				_pTimeValue := F_BACnet_EndOf(_pDailySched, SIZEOF(ST_BACnet_SpecialEventList));
				_nTimeValue := 1;
				WHILE _pTimeValue <> 0 DO
					Sched_ReadEntry(eDatatype, _pTimeValue, tCalendar[_nCalEntry].stEntry[_nTimeValue]);
					_nTimeValue:=_nTimeValue+1;
					_pTimeValue:=F_BACnet_NextListElem(_pTimeValue, _pTimeValue^.nEntrySize);
				END_WHILE		
				_nCalEntry:=_nCalEntry+1;
			ELSE
				tException[_nExcEntry].eType := _pDailySched^.stEvent.eCalEntryChoice + 1;
				tException[_nExcEntry].uDate := _pDailySched^.stEvent.uCalEntry;
				tException[_nExcEntry].nEventPriority := _pDailySched^.stEvent.nEventPriority;
				
				_pTimeValue := F_BACnet_EndOf(_pDailySched, SIZEOF(ST_BACnet_SpecialEventList));
				_nTimeValue := 1;
				WHILE _pTimeValue <> 0 DO
					Sched_ReadEntry(eDatatype, _pTimeValue, tException[_nExcEntry].stEntry[_nTimeValue]);
					_nTimeValue:=_nTimeValue+1;
					_pTimeValue:=F_BACnet_NextListElem(_pTimeValue, _pTimeValue^.nEntrySize);
				END_WHILE					
				_nExcEntry:=_nExcEntry+1;
			END_IF
			_pDailySched:=F_BACnet_NextListElem(_pDailySched, _pDailySched^.nEntrySize);
		END_WHILE
	END_IF
END_IF

ReadPropertyExceptionSched:=_hResult;
END_METHOD

METHOD ReadPropertyLimitEnable : HRESULT
VAR CONSTANT
	ePropID : E_BACnetPropIdentifier := E_BACnetPropIdentifier.PropLimitEnable;
END_VAR
VAR_INPUT
	value : REFERENCE TO ST_BACnet_LimitEnable;
END_VAR
VAR
	_flags : WORD := 16#0006;
	_size : DINT := 2;
END_VAR
IF (ipObj <> 0) AND (__ISVALIDREF(value)) THEN
	ReadPropertyLimitEnable := ReadProperty(ePropID, ADR(_flags), ADR(_size));
	
	IF (ReadPropertyLimitEnable = S_OK) THEN
		value.highLimitEnable := _flags.14;
		value.lowLimitEnable := _flags.15;
	END_IF
ELSE
	ReadPropertyLimitEnable := E_FAIL;
END_IF
END_METHOD

METHOD ReadPropertyLogBuffer : HRESULT
VAR_IN_OUT
	tLogBuffer						: ARRAY [*] OF ST_BA_TrendEntry;
END_VAR
VAR
	_nLength						: DINT;
	_cbTotalBuf						: UDINT;
	
	_pLbRecordList					: POINTER TO ST_BACnet_LogRecordList;								// Log buffer - record list
	_pLrDatumList					: POINTER TO ST_BACnet_LogDatumList;
	_nNextRecPos					: UDINT;
	_nRecCount						: UDINT;															// Log record entry - datum list
	_nMaxSeq						: DWORD;
	
	_nRec							: UDINT;
	
	
	_stRecListTmp					: POINTER TO ST_BACnet_LogRecordList;
END_VAR
IF (ipObj = 0) THEN
	_hResult := E_FAIL;
ELSE
	_nLength := SIZEOF(BACnet_Globals.bDefaultBuffer);
	_hResult := ReadProperty(E_BACnetPropIdentifier.PropLogBuffer, ADR(BACnet_Globals.bDefaultBuffer), ADR(_nLength));
	
	IF (SUCCEEDED(_hResult)) THEN
		IF (_nLength > 0) THEN
			MEMSET(ADR(tLogBuffer), 0, TO_UDINT(F_BA_TrendBufferSize(tLogBuffer)));
			
			// Point to first data:
			_pLbRecordList := ADR(BACnet_Globals.bDefaultBuffer);
			_cbTotalBuf := 0;
			_nNextRecPos := 0;
			_nRecCount := 0;
			_nMaxSeq := 0;
			
			REPEAT
				IF ((_pLbRecordList^.nEntrySize AND 16#7FFFFFFF) > 0) THEN
	
					_stRecListTmp := _pLbRecordList;
					
(* DEBUG *)			iOwner.LogMsg.Show3(ADSLOG_MSGTYPE_ERROR, 'DBG_TLOG', 'Record= %d, SeqID=%d, Size=%d', F_UDINT(_nNextRecPos), F_UDINT(_stRecListTmp^.nSequence), F_UDINT(_stRecListTmp^.nEntrySize), TRUE);
		
		
					(*
					// Insert pointer to record entry:
					_arrRecords[_nNextRecPos] := _pLbRecordList;
					*)
					// Select next free record position and count:
					_nNextRecPos := _nNextRecPos + 1;
					_nRecCount := _nRecCount + 1;
				END_IF
	
				// Next record entry:
				IF (NOT Trend_NextLogRecord(_pLbRecordList, _cbTotalBuf)) THEN
					EXIT;
				END_IF

			UNTIL (		(_nRecCount >= (BACnet_Globals.nDataField_MaxLogBufferEntries+1)) (* result buffer full *)
					OR	(_pLbRecordList >= (ADR(BACnet_Globals.bDefaultBuffer) + _nLength)) (* ads buffer ending reached *)
				)
			END_REPEAT

			
(* DEBUG *)	iOwner.LogMsg.Show(ADSLOG_MSGTYPE_ERROR, 'DBG_TLOG', '-----------------', TRUE);

//			// Select record list entry:
//			REPEAT
//				IF ((_pLbRecordList^.nEntrySize AND 16#7FFFFFFF) > 0) THEN
//	
//					(* check sequence order *)
//					IF _nMaxSeq > _pLbRecordList^.nSequence THEN
//						(* current sequence is lower then previous one - scan entries and sort *)
//						FOR _nRec := 0 TO _nRecCount-1 DO
//							IF _arrRecords[_nRec]^.nSequence > _pLbRecordList^.nSequence THEN
//								(* found higher sequence no. - move *)
//								_nNextRecPos := _nRec; (* remind insert position *)
//								(* check free space *)
//								IF (_nRecCount-1 < BACnet_Globals.nDataField_MaxLogBufferEntries) THEN
//									(* enough space at end of list - move *)
//									MEMMOVE(	ADR(_arrRecords[_nRec+1]), (* one position up *)
//												ADR(_arrRecords[_nRec]), (* free insert position *)
//												(_nRecCount - _nRec)*SIZEOF(_arrRecords[0]) (* move all element behind insert position *)
//									);
//								END_IF
//								EXIT; (* leave *)
//							END_IF
//						END_FOR
//					ELSE
//						(* remind sequence no. *)
//						_nMaxSeq := _pLbRecordList^.nSequence;
//					END_IF
//	
//					(* insert pointer to record entry *)
//					_arrRecords[_nNextRecPos] := _pLbRecordList;
//					(* select next free record position and count *)
//					_nNextRecPos := _nNextRecPos + 1;
//					_nRecCount := _nRecCount + 1;
//				END_IF
//	
//				(* next record entry *)
//				_NextLogRecord();
//	
//			UNTIL (		(NOT _bNextRecord) (* no more record entries *)
//					OR	(_nRecCount >= (BACnet_Globals.nDataField_MaxLogBufferEntries+1)) (* result buffer full *)
//					OR	(_pLbRecordList >= (_pAdsBuf + stBACnet_AdsBuffer.iLocked)) (* ads buffer ending reached *)
//				)
//			END_REPEAT
			
		END_IF
	ELSE
		iOwner.LogMsg.Show1(ADSLOG_MSGTYPE_ERROR, 'RLB23', 'Failed to read log buffer property! (Error 0x%x)', F_DINT(_hResult), TRUE);
	END_IF
END_IF


ReadPropertyLogBuffer := _hResult;
END_METHOD

METHOD ReadPropertyNotifyType : HRESULT
VAR CONSTANT
	ePropID : E_BACnetPropIdentifier := E_BACnetPropIdentifier.PropNotifyType;
END_VAR
VAR_INPUT
	value : REFERENCE TO E_BACnet_NotifyType;
END_VAR
VAR
	_size : DINT := 4;
END_VAR
IF (ipObj <> 0) AND (__ISVALIDREF(value)) THEN
	ReadPropertyNotifyType := ReadProperty(ePropID, ADR(value), ADR(_size));
ELSE
	ReadPropertyNotifyType := E_FAIL;
END_IF
END_METHOD

METHOD ReadPropertyReal : HRESULT
VAR_INPUT
	ePropID : E_BACnetPropIdentifier;
	value : REFERENCE TO REAL;
END_VAR
VAR
	_size : DINT := 4;
END_VAR
IF (ipObj <> 0) AND (__ISVALIDREF(value)) THEN
	ReadPropertyReal := ReadProperty(ePropID, ADR(value), ADR(_size));
ELSE
	ReadPropertyReal := E_FAIL;
END_IF
END_METHOD

METHOD ReadPropertyRecipientList : HRESULT
VAR_IN_OUT
	stRecipientList			: ARRAY[*] OF ST_BACnet_Destination;
END_VAR
// [Bugworkaround]
// > _stUnused" has to be static, otherwise its memory can be initialized incorrectly by PLC :(
VAR_STAT
	_nTemp					: DINT;
	_nSize					: DINT;
	_stUnused				: ST_BACnet_Destination;
END_VAR
IF (ipObj = 0) THEN
	_hResult := E_FAIL;
ELSE
	// Reset current content:
	F_BA_MemSetArr(stRecipientList, LOWER_BOUND(stRecipientList, 1), UPPER_BOUND(stRecipientList, 1), _stUnused);
		
	_nSize := (UPPER_BOUND(stRecipientList, 1) - LOWER_BOUND(stRecipientList, 1) + 1) * SIZEOF(ST_BACnet_Destination);
	_hResult := ReadProperty(E_BACnetPropIdentifier.PropRecipientList, stRecipientList, ADR(_nSize));
END_IF

ReadPropertyRecipientList := _hResult;
END_METHOD

METHOD ReadPropertyReference : HRESULT
VAR_INPUT
	eProperty				: E_BACnetPropIdentifier;
END_VAR
VAR_IN_OUT
	stRefObject				: ST_BACnet_ObjectPropertyReference;
END_VAR
VAR
	stTemp					: ST_BACnet_DeviceObjectPropertyReference;
END_VAR
IF (ipObj <> 0) THEN
	ReadPropertyReference := ReadProperty(eProperty, ADR(stTemp), ADR(stTemp));
	
	IF (S_OK = ReadPropertyReference) THEN
		stRefObject.tObjectID := stTemp.tObjId;
		stRefObject.ePropertyId := stTemp.ePropIdentifier;
	
		// Reset previous reference.
		// > Current interface pointer has to be resolved now via PLC!
		stRefObject.iObject := 0;
	END_IF
ELSE
	ReadPropertyReference := E_FAIL;
END_IF
END_METHOD

METHOD ReadPropertyStatusFlags : HRESULT
VAR_INPUT
	stateFlags : REFERENCE TO ST_BA_StatusFlags;
END_VAR
VAR
	_flags : DWORD;
	_size : DINT := 2;
END_VAR
IF (ipObj <> 0) AND (__ISVALIDREF(stateFlags)) THEN
	ReadPropertyStatusFlags:=ReadProperty(E_BACnetPropIdentifier.PropStatusFlags, ADR(_flags), ADR(_size));
	
	IF (ReadPropertyStatusFlags = S_OK) THEN
		stateFlags.bInAlarm:= F_BACnet_IsBitFieldBitSet(_flags, E_BACnet_StatusFlags.eInAlarm);
		stateFlags.bFault:= F_BACnet_IsBitFieldBitSet(_flags, E_BACnet_StatusFlags.eFault);
		stateFlags.bOverridden:= F_BACnet_IsBitFieldBitSet(_flags, E_BACnet_StatusFlags.eOverridden);
		stateFlags.bOutOfService:= F_BACnet_IsBitFieldBitSet(_flags, E_BACnet_StatusFlags.eOutOfService);
	END_IF
ELSE
	ReadPropertyStatusFlags := E_FAIL;
END_IF
END_METHOD

METHOD ReadPropertyString : HRESULT
VAR_INPUT
	ePropID : E_BACnetPropIdentifier;
	value : REFERENCE TO T_MaxString;
END_VAR
VAR
	_size : UDINT := 255;
	_fbDecode : FB_BACnet_StringExtDecode;
END_VAR
IF (ipObj <> 0) AND (__ISVALIDREF(value)) THEN
	_size:=SIZEOF(BACnet_Globals.stADSBuffer);
	ReadPropertyString:=ReadProperty(ePropID, ADR(BACnet_Globals.stADSBuffer), ADR(_size));
	
	IF (ReadPropertyString = S_OK) THEN
		memset(ADR(value)+_size,0,1);
		_fbDecode(pChrStringExt:=ADR(BACnet_Globals.stADSBuffer), pOutString:=ADR(value), nOutSize:=_size);
		
		IF NOT _fbDecode.bValid THEN
			ReadPropertyString := E_FAIL;	
		END_IF
	END_IF
ELSE
	ReadPropertyString := E_FAIL;
END_IF
END_METHOD

METHOD ReadPropertyUDInt : HRESULT
VAR_INPUT
	ePropID : E_BACnetPropIdentifier;
	value : REFERENCE TO UDINT;
END_VAR
VAR
	_size : DINT := 4;
END_VAR
IF (ipObj <> 0) AND (__ISVALIDREF(value)) THEN
	ReadPropertyUDInt := ReadProperty(ePropID, ADR(value), ADR(_size));
ELSE
	ReadPropertyUDInt := E_FAIL;
END_IF
END_METHOD

METHOD ReadPropertyUnit : HRESULT
VAR CONSTANT
	ePropID : E_BACnetPropIdentifier := E_BACnetPropIdentifier.PropUnits;
END_VAR
VAR_INPUT
	value : REFERENCE TO E_BA_Unit;
END_VAR
VAR
	_size : DINT := 4;
END_VAR
IF (ipObj <> 0) AND (__ISVALIDREF(value)) THEN
	ReadPropertyUnit := ReadProperty(ePropID, ADR(value), ADR(_size));
ELSE
	ReadPropertyUnit := E_FAIL;
END_IF
END_METHOD

METHOD ReadPropertyWeeklySched : HRESULT
VAR_IN_OUT
	stWeek							: ARRAY[*, *] OF ST_BA_SchedEntry;
END_VAR
VAR_INPUT
	eDatatype						: E_BACnet_ValueChoice;
END_VAR
VAR			
	// General:
	nLenTmp							: UDINT;
	nLength							: DINT;
	
	_cbTmpSize						: UDINT;
	_cbTotalEntry					: UDINT;
	_cbTotalBuf						: UDINT;
	
	// Scheduler:
	_pDailySched					: POINTER TO ST_BACnet_DailySchedule;
	_pTimeValue						: POINTER TO ST_BACnet_TimeValueList;
	_pOldTimeValue					: POINTER TO ST_BACnet_TimeValueList;
	_nDayTmp						: DINT;
	_nDayEntryTmp					: DINT;
	_nDays							: UINT;
END_VAR
IF (ipObj = 0) THEN
	_hResult := E_FAIL;
	
ELSIF (eDataType = E_BACnet_ValueChoice.eNullValue) THEN
	iOwner.LogMsg.Show(ADSLOG_MSGTYPE_ERROR, 'RWS05', 'Invalid datatype!', TRUE);
	_hResult := E_FAIL;
ELSE
	nLength := SIZEOF(BACnet_Globals.bDefaultBuffer);
	_hResult := ReadProperty(E_BACnetPropIdentifier.PropWeeklySchedule, ADR(BACnet_Globals.bDefaultBuffer), ADR(nLength));
	
	IF (SUCCEEDED(_hResult)) THEN
		IF (nLength > 0) THEN
			// Clear content:
			_nDayTmp := F_BA_WeeklySchedSize(stWeek);
			MEMSET(stWeek, 0, TO_UDINT(F_BA_WeeklySchedSize(stWeek)));
			
			// Point to first data:
			_pDailySched := ADR(BACnet_Globals.bDefaultBuffer);
			_pTimeValue := ADR(_pDailySched^.stListEntry);
			_nDayEntryTmp := LOWER_BOUND(stWeek, 2);
			_nDayTmp := LOWER_BOUND(stWeek, 1);
			
			WHILE (_pTimeValue <> 0) AND SUCCEEDED(_hResult) DO
				(* check entry size of time value *)
				IF (_pTimeValue^.nEntrySize AND 16#7FFFFFFF) > 0 THEN
					(* check internal schedule buffer index *)
					IF (_nDayTmp > E_BA_Weekday.eSunday) THEN
						iOwner.LogMsg.Show(ADSLOG_MSGTYPE_ERROR, 'RWS23', 'Wrong day index!', TRUE);
						_hResult := E_FAIL;
					ELSE
						IF (_nDayEntryTmp <= TO_INT(BACnet_Globals.nDataField_MaxDayEntry)) THEN
							Sched_ReadEntry(eDatatype, _pTimeValue, stWeek[_nDayTmp, _nDayEntryTmp]);							
							_nDayEntryTmp := _nDayEntryTmp + 1;
						ELSE
							iOwner.LogMsg.Show(ADSLOG_MSGTYPE_WARN, 'RWS74', 'Max. count of entries reached!', TRUE);
						END_IF
	
						(* next time value entry *)
						(* check if next time value entry available *)
						IF (NOT Sched_SetNextTimeVal(_pDailySched, _pTimeValue, _cbTmpSize, _pOldTimeValue)) THEN
							(* update pointer each cycle (even if no day follows!) *)
							(* check for next day *)
							IF (NOT Sched_SetNextDay(_pDailySched, _cbTmpSize, _cbTotalBuf, _pOldTimeValue, _nDayTmp, _nDayEntryTmp, _pTimeValue)) THEN
								// Job done!
								EXIT;
							END_IF
						END_IF
					END_IF
	
				ELSE
					(* update pointer each cycle (even if no day follows!) *)
					(* No timevalue entry, check if next day element exists and pointer is plausible *)
					IF (Sched_SetNextDay(_pDailySched, _cbTmpSize, _cbTotalBuf, _pOldTimeValue, _nDayTmp, _nDayEntryTmp, _pTimeValue)) THEN
						
						// Check pointer:
						IF (_pDailySched + (_pDailySched^.nEntrySize AND 16#7FFFFFFF)) >= (ADR(BACnet_Globals.bDefaultBuffer) + SIZEOF(BACnet_Globals.bDefaultBuffer)) THEN
							iOwner.LogMsg.Show(ADSLOG_MSGTYPE_ERROR, 'RWS96', 'Insufficient buffer size!', TRUE);
							_hResult := E_FAIL;
						END_IF
					ELSE
						// Job done!
						EXIT;
					END_IF
				END_IF
				
				// Check bounds:
				IF (_nDayTmp > UPPER_BOUND(stWeek, 1)) OR (_nDayEntryTmp > UPPER_BOUND(stWeek, 2)) THEN
					EXIT;
				END_IF
			END_WHILE
		END_IF
	END_IF
END_IF

ReadPropertyWeeklySched := _hResult;
END_METHOD

METHOD INTERNAL GetSyncHandleMode : BOOL
VAR_INPUT
	eMode		: E_BA_FullSyncMode;
END_VAR
VAR_OUTPUT
	eResult		: E_BA_SyncMode;
END_VAR
CASE (eMode) OF
	eSync_FromSupplement:
		eResult := E_BA_SyncMode.eFromSupplement;
		
	eSync_ToSupplement,
	eFullSync_InitSupplement,
	eFullSync_InitPLC:
		eResult := E_BA_SyncMode.eToSupplement;
ELSE
	eResult := E_BA_SyncMode.eNone;
END_CASE

GetSyncHandleMode := (eResult <> E_BA_SyncMode.eNone);
END_METHOD

METHOD PRIVATE AddListElement : BOOL
VAR_INPUT
	ePropID				: E_BACnetPropIdentifier;
	nIndex				: DINT;
	nSize				: DINT;
	pValue				: PVOID;
END_VAR
VAR
	nListLen			: DINT;
	_size				: DINT := SIZEOF(DINT);
END_VAR
// Read current element count:
IF ipObj.SyncReadProperty(ePropID, ADR(nListLen), ADR(_size), 0) = S_OK THEN
	IF nListLen < nIndex THEN
		// Add new element to list:
		AddListElement := (ipObj.SyncWriteProperty(ePropID, pValue, nSize, 16#FFFFFFFE) = S_OK);
	ELSE
		AddListElement := TRUE;
	END_IF
END_IF
END_METHOD

METHOD PRIVATE ApplySyncHandler : BOOL
VAR
	_i		: E_BA_SyncMode;
END_VAR
ApplySyncHandler := TRUE;

// Apply requested sync handlers:
FOR _i := E_BA_SyncMode.eFromSupplement TO E_BA_SyncMode.eToSupplement DO
	IF (nReqSyncHandlers[_i] > 0) THEN
		IF (NOT SetPropertyCount(nReqSyncHandlers[_i], _i)) THEN
			ApplySyncHandler := FALSE;
		END_IF
	END_IF
END_FOR
END_METHOD

METHOD PRIVATE EvaluatePropSync
VAR_INPUT
	hResult		: HRESULT;
	eSyncMode	: E_BA_FullSyncMode;
	bCyclic		: BOOL := FALSE;
END_VAR
VAR
	_eMode		: E_BA_SyncMode	:= E_BA_SyncMode.eNone;
END_VAR
IF SUCCEEDED(hResult) THEN
	// Cyclic property synchronization:
	IF ((bCyclic) AND (eSyncMode > eSync_FromSupplement)) THEN
		nCycPropCnt := (nCycPropCnt+1);
	END_IF
	
	// Increment SyncHandlers:
	IF (GetSyncHandleMode(eSyncMode, eResult=>_eMode)) THEN
		nSyncHandlers[_eMode] := (nSyncHandlers[_eMode]+1);
	END_IF
END_IF
END_METHOD

METHOD RequestSyncHandlers : BOOL
VAR_INPUT
	nFromSupplement		: UDINT		:= 0;
	nToSupplement		: UDINT		:= 0;
END_VAR
nReqSyncHandlers[E_BA_SyncMode.eFromSupplement] := (nReqSyncHandlers[E_BA_SyncMode.eFromSupplement]+nFromSupplement);
nReqSyncHandlers[E_BA_SyncMode.eToSupplement] := (nReqSyncHandlers[E_BA_SyncMode.eToSupplement]+nToSupplement);
END_METHOD

METHOD RequestSyncHandlersEx : BOOL
VAR_INPUT
	eMode		: E_BA_FullSyncMode;
	nCount		: UDINT		:= 0;
END_VAR
VAR
	_eMode		: E_BA_SyncMode	:= E_BA_SyncMode.eNone;
END_VAR
IF (GetSyncHandleMode(eMode, eResult=>_eMode)) THEN
	nReqSyncHandlers[_eMode] := (nReqSyncHandlers[_eMode]+nCount);
	
	RequestSyncHandlersEx := TRUE;
END_IF
END_METHOD

METHOD SyncProperty : HRESULT
VAR_INPUT
	ePropID : E_BACnetPropIdentifier;
	nSize : UDINT;
	pValue : PVOID;
	pData : PVOID := 0;
	eSyncMode : E_BA_FullSyncMode;
	bCyclic : BOOL := FALSE;
END_VAR
VAR
	nIndex : UDINT := 16#FFFFFFFF;
END_VAR
_hResult := SEL(Error, ipObj.SyncPropertyData(ePropID, nSize, pValue, pData, 0, nIndex, TO_UINT(eSyncMode)), E_FAIL);
SyncProperty:=_hResult;

EvaluatePropSync(_hResult, eSyncMode, bCyclic);
END_METHOD

METHOD SyncPropertyCOV : BOOL
VAR_IN_OUT
	bChangeTrig : BOOL;
END_VAR
VAR_INPUT
	ePropertyID : E_BACnetPropIdentifier;
END_VAR
VAR
	_hResult : HRESULT;
END_VAR
// Initialize COV-Trigger:
_hResult := SyncProperty(ePropertyID, 0, 0, ADR(bChangeTrig), eSync_FromSupplement, FALSE);
IF (_hResult <> S_OK) THEN
	iOwner.LogMsg.Show2(ADSLOG_MSGTYPE_ERROR, 'SPCOV03', 'Initialize COV-Trigger of property "%d" failed (Error: "0x%x")!', F_INT(ePropertyID), F_DINT(_hResult), TRUE);
ELSE
	SyncPropertyCOV := TRUE;
	bChangeTrig := FALSE;
END_IF
END_METHOD

METHOD SyncPropertyIdx : HRESULT
VAR_INPUT
	ePropID : E_BACnetPropIdentifier;
	nSize : UDINT;
	pValue : PVOID;
	nIndex : INT := -1;
	pData : PVOID := 0;
	eSyncMode : E_BA_FullSyncMode;
	bCyclic : BOOL := FALSE;
END_VAR
SyncPropertyIdx := SEL(Error, ipObj.SyncPropertyData(ePropID, nSize, pValue, pData, 0, TO_UDINT(nIndex), TO_UINT(eSyncMode)), E_FAIL);

EvaluatePropSync(_hResult, eSyncMode, bCyclic);
END_METHOD

METHOD SyncPropertyList : BOOL
VAR_INPUT
	ePropID				: E_BACnetPropIdentifier;
	pList				: PVOID;
	nItemSize			: UDINT;
	nItemCount			: UDINT;
	eSyncMode			: E_BA_FullSyncMode;
	bValidate			: BOOL						:= FALSE;			// Check items contents and stops synchronization if an used items is found.
END_VAR
VAR
	_nTemp				: UDINT;
	_pValue				: PVOID;
END_VAR
IF (bValidate) THEN
	RemoveListElements(ePropID);
END_IF

IF (pList <> 0) AND (nItemSize > 0) AND (nItemCount > 0) THEN
	FOR _nTemp := 1 TO nItemCount DO
		_pValue := (pList + ((_nTemp-1) * nItemSize));
		
		IF (bValidate) AND_THEN (F_BA_ByteCmp(_pValue, nItemSize, 0) = 0) THEN
			// Synchronization of used items completed:
			EXIT;
		END_IF
	
		IF NOT AddListElement(ePropID, TO_DINT(_nTemp), SIZEOF(STRING), _pValue) THEN
			RETURN;
		ELSIF SyncPropertyIdx(ePropID, SIZEOF(STRING), _pValue, TO_INT(_nTemp), 0, eSyncMode, FALSE) <> S_OK THEN
			RETURN;
		END_IF
	END_FOR
	
	SyncPropertyList := TRUE;
END_IF
END_METHOD

METHOD SyncPropertyPvPrio : HRESULT
VAR_INPUT
	ePropID : E_BACnetPropIdentifier;
	nSize : UDINT;
	pValue : PVOID;
	bEnPriority : POINTER TO BOOL;
	nPriority : UDINT := 16#FFFFFFFF;
	pData : PVOID := 0;
	eSyncMode : E_BA_FullSyncMode;
	bCyclic : BOOL := FALSE;
END_VAR
SyncPropertyPvPrio := SEL(Error, ipObj.SyncPropertyData(ePropID, nSize, pValue, pData, bEnPriority, nPriority, TO_UINT(eSyncMode)), E_FAIL);

EvaluatePropSync(_hResult, eSyncMode, bCyclic);
END_METHOD

METHOD WriteProperty : HRESULT
VAR_INPUT
	ePropID : E_BACnetPropIdentifier;
	pData : PVOID;
	nData : DINT;
END_VAR
IF (ipObj <> 0) THEN
	WriteProperty:=ipObj.SyncWriteProperty(TO_INT(ePropID), pData, nData, 16#FFFFFFFF);
	
	IF (WriteProperty <> S_OK) THEN
		iOwner.LogMsg.Show2(ADSLOG_MSGTYPE_ERROR, 'WP5', 'Writing property "%d" failed (Error "0x%x")!', F_INT(ePropID), F_DINT(WriteProperty), TRUE);
	END_IF
ELSE
	WriteProperty := E_FAIL;
END_IF
END_METHOD

METHOD WritePropertyBool : HRESULT
VAR_INPUT
	ePropID : E_BACnetPropIdentifier;
	bValue : BOOL;
END_VAR
IF (ipObj <> 0) THEN
	WritePropertyBool := WriteProperty(ePropID, ADR(bValue), SIZEOF(bValue));
ELSE
	WritePropertyBool := E_FAIL;
END_IF
END_METHOD

METHOD WritePropertyDateList : HRESULT
VAR_IN_OUT
	stDateList				: ARRAY[*] OF ST_BA_CalendarEntry;
END_VAR
VAR
	_i						: DINT;
	
	_stEntry				: POINTER TO ST_BACnet_CalendarEntry;
	_cbTotalBuf				: UDINT;
END_VAR
IF (ipObj = 0) THEN
	_hResult := E_FAIL;
ELSE
	_stEntry := ADR(BACnet_Globals.bDefaultBuffer);
	_cbTotalBuf := 0;
	
	FOR _i := LOWER_BOUND(stDateList, 1) TO UPPER_BOUND(stDateList, 1) DO
		IF (F_BACnet_ToDateListEntry(ADR(stDateList[_i]), stResult=>_stEntry^)) THEN		
			_stEntry := (_stEntry+SIZEOF(ST_BACnet_CalendarEntry));
			_cbTotalBuf := (_cbTotalBuf+SIZEOF(ST_BACnet_CalendarEntry));
		END_IF
	END_FOR
	
	// Write data:
	_hResult := WriteProperty(E_BACnetPropIdentifier.PropDateList, ADR(BACnet_Globals.bDefaultBuffer), TO_DINT(_cbTotalBuf));
END_IF	

WritePropertyDateList := _hResult;
END_METHOD

METHOD WritePropertyEventEnable : HRESULT
VAR_INPUT
	bToNormal : BOOL;
	bToFault : BOOL;
	bToOffNormal : BOOL;
END_VAR
VAR
	_flags : WORD := 16#0005;
END_VAR
IF (ipObj <> 0) THEN
	IF bToNormal THEN
		_flags:=_flags OR 16#2000;
	END_IF
	IF bToFault THEN
		_flags:=_flags OR 16#4000;
	END_IF
	IF bToOffNormal THEN
		_flags:=_flags OR 16#8000;
	END_IF

	WritePropertyEventEnable := WriteProperty(E_BACnetPropIdentifier.PropEventEnable, ADR(_flags), 2);
ELSE
	WritePropertyEventEnable := E_FAIL;
END_IF
END_METHOD

METHOD WritePropertyExceptionSched : HRESULT
VAR_IN_OUT
	tCalendar			: T_BACnet_SchedCalendar;
	tException			: T_BACnet_SchedExceptionList;
END_VAR
VAR_INPUT
	eDatatype			: E_BACnet_ValueChoice;
END_VAR
VAR
	_nEntry				: INT;
	_nSchedEntry		: INT;
	_hResult			: HRESULT;
	_pDailySched		: POINTER TO ST_BACnet_SpecialEventList;
	_pDailySchedOld		: POINTER TO ST_BACnet_SpecialEventList;
	_cbTotalSize		: UDINT;
	_cbTmpSize			: UDINT;
	_calObjId 			: T_BACnet_ObjectIdentifier;
	_pTimeValue			: POINTER TO ST_BACnet_TimeValueList;
	_pOldTimeValue		: POINTER TO ST_BACnet_TimeValueList;
END_VAR
IF ipObj = 0 THEN
	_hResult := E_FAIL;
ELSE
	_pDailySched := ADR(BACnet_Globals.bDefaultBuffer);
	_pDailySchedOld := 0;
	_cbTotalSize := 0;
	
	FOR _nEntry:=1 TO BACnet_Param.nSched_CalendarCount DO
		IF F_BACnet_IsObjIdentifierValid(tCalendar[_nEntry].tRefCalendarID) THEN
			MEMSET(ADR(_pDailySched^.stEvent), 0, SIZEOF(_pDailySched^.stEvent));
			_pDailySched^.nEntrySize := SIZEOF(_pDailySched^.stEvent);
			_pDailySched^.nRes := 0;
			_pDailySched^.stEvent.eEventChoice := E_BACnet_SpecialEventChoice.eCalendarReference;
			_pDailySched^.stEvent.nEventPriority := SEL(F_BACnet_IsPriorityValid(tCalendar[_nEntry].eEventPriority), 1, TO_UDINT(tCalendar[_nEntry].eEventPriority));
				
			IF  _pDailySchedOld <> 0 THEN
				_pDailySchedOld^.nEntrySize := _pDailySchedOld^.nEntrySize + 16#80000000;
			END_IF
			
			_calObjId := tCalendar[_nEntry].tRefCalendarID;
			MEMCPY(ADR(_pDailySched^.stEvent.eCalEntryChoice), ADR(_calObjId), SIZEOF(_calObjId));
			
			_pOldTimeValue := 0;
			_pTimeValue:= F_BACnet_EndOf(_pDailySched, SIZEOF(ST_BACnet_SpecialEventList));
			FOR _nSchedEntry:=1 TO BACnet_Param.nSched_EntryCount DO
				 IF tCalendar[_nEntry].stEntry[_nSchedEntry].eState = E_BA_SchedEntryState.eValue THEN 
					 _pTimeValue^.nEntrySize := 0;
					 _pTimeValue^.nRes := 0;
					 
					 // Set flag "next entry" to the previous element:
					IF (_nSchedEntry > 1) AND (_pOldTimeValue <> 0) THEN
						_pOldTimeValue^.nEntrySize := _pOldTimeValue^.nEntrySize + 16#80000000;
					END_IF
					
					Sched_WriteEntry(eDatatype, _pTimeValue, tCalendar[_nEntry].stEntry[_nSchedEntry]); 
					
					_pDailySched^.nEntrySize := _pDailySched^.nEntrySize + _pTimeValue^.nEntrySize + SIZEOF(_pTimeValue^.nEntrySize) + SIZEOF(_pTimeValue^.nRes);	
										
					_pOldTimeValue := _pTimeValue;
					_pTimeValue := _pTimeValue +  F_BACnet_AlignedSize(_pTimeValue^.nEntrySize AND 16#7FFFFFFF) + SIZEOF(_pTimeValue^.nEntrySize) + SIZEOF(_pTimeValue^.nRes);					 
				 END_IF
			END_FOR
		
			_cbTotalSize := _cbTotalSize + _pDailySched^.nEntrySize + SIZEOF(_pDailySched^.nEntrySize) + SIZEOF(_pDailySched^.nRes);	
			_pDailySchedOld := _pDailySched;
			_pDailySched := _pDailySched +  F_BACnet_AlignedSize(_pDailySched^.nEntrySize AND 16#7FFFFFFF) + SIZEOF(_pDailySched^.nEntrySize) + SIZEOF(_pDailySched^.nRes);					 		
		END_IF
	END_FOR
	
	FOR _nEntry:=1 TO BACnet_Param.nSched_ExceptionCount DO
		IF tException[_nEntry].eType <> E_BA_DateValChoice.Invalid THEN
			MEMSET(ADR(_pDailySched^.stEvent), 0, SIZEOF(_pDailySched^.stEvent));
			_pDailySched^.nEntrySize := SIZEOF(_pDailySched^.stEvent);
			_pDailySched^.nRes := 0;
			_pDailySched^.stEvent.eEventChoice := E_BACnet_SpecialEventChoice.eCalendarEntry;
			IF tException[_nEntry].nEventPriority > 0 AND tException[_nEntry].nEventPriority < 17 THEN
				_pDailySched^.stEvent.nEventPriority := tException[_nEntry].nEventPriority; 
			ELSE
				_pDailySched^.stEvent.nEventPriority := 1;
			END_IF
			IF _pDailySchedOld <> 0 THEN
				_pDailySchedOld^.nEntrySize := _pDailySchedOld^.nEntrySize + 16#80000000;
			END_IF
			
			_pDailySched^.stEvent.eCalEntryChoice := tException[_nEntry].eType-1;
			_pDailySched^.stEvent.uCalEntry := tException[_nEntry].uDate;
			
			_pOldTimeValue := 0;
			_pTimeValue:= F_BACnet_EndOf(_pDailySched, SIZEOF(ST_BACnet_SpecialEventList));
			FOR _nSchedEntry:=1 TO BACnet_Param.nSched_EntryCount DO
				CASE (tException[_nEntry].stEntry[_nSchedEntry].eState) OF
					E_BA_SchedEntryState.eNull,
					E_BA_SchedEntryState.eValue:
						 _pTimeValue^.nEntrySize := 0;
						 _pTimeValue^.nRes := 0;
						 
						 // Set flag "next entry" to the previous element:
						IF (_nSchedEntry > 1) AND (_pOldTimeValue <> 0) THEN
							_pOldTimeValue^.nEntrySize := _pOldTimeValue^.nEntrySize + 16#80000000;
						END_IF
						
						Sched_WriteEntry(eDatatype, _pTimeValue, tException[_nEntry].stEntry[_nSchedEntry]); 
						
						_pDailySched^.nEntrySize := _pDailySched^.nEntrySize + _pTimeValue^.nEntrySize + SIZEOF(_pTimeValue^.nEntrySize) + SIZEOF(_pTimeValue^.nRes);	
											
						_pOldTimeValue := _pTimeValue;
						_pTimeValue := _pTimeValue +  F_BACnet_AlignedSize(_pTimeValue^.nEntrySize AND 16#7FFFFFFF) + SIZEOF(_pTimeValue^.nEntrySize) + SIZEOF(_pTimeValue^.nRes);					 
				END_CASE
			END_FOR
				
			_cbTotalSize := _cbTotalSize + _pDailySched^.nEntrySize + SIZEOF(_pDailySched^.nEntrySize) + SIZEOF(_pDailySched^.nRes);	
			_pDailySchedOld := _pDailySched;
			_pDailySched := _pDailySched +  F_BACnet_AlignedSize(_pDailySched^.nEntrySize AND 16#7FFFFFFF) + SIZEOF(_pDailySched^.nEntrySize) + SIZEOF(_pDailySched^.nRes);					 
		END_IF
	END_FOR
	
	IF (_cbTotalSize = 0) THEN
		// Indicate empty exception property:
		_cbTotalSize := 8;
		MEMSET(ADR(BACnet_Globals.bDefaultBuffer), 0, _cbTotalSize);
	END_IF
	
	// Write data:
	_hResult := WriteProperty(E_BACnetPropIdentifier.PropExceptionSchedule, ADR(BACnet_Globals.bDefaultBuffer), TO_DINT(_cbTotalSize));
END_IF

WritePropertyExceptionSched := _hResult;
END_METHOD

METHOD WritePropertyLimitEnable : HRESULT
VAR_INPUT
	bLowLimitEnable : BOOL;
	bHighLimitEnable : BOOL;
END_VAR
VAR
	_flags : WORD := 16#0006;
END_VAR
IF (ipObj <> 0) THEN
	IF bLowLimitEnable THEN
		_flags:=_flags OR 16#8000;
	END_IF
	IF bHighLimitEnable THEN
		_flags:=_flags OR 16#4000;
	END_IF

	WritePropertyLimitEnable := WriteProperty(E_BACnetPropIdentifier.PropLimitEnable, ADR(_flags), 2);
ELSE
	WritePropertyLimitEnable := E_FAIL;
END_IF
END_METHOD

METHOD WritePropertyLogBuffer : HRESULT
VAR_IN_OUT
	tLogBuffer						: ARRAY [*] OF ST_BA_TrendEntry;
END_VAR
IF (ipObj = 0) THEN
	_hResult := E_FAIL;
ELSE
	_hResult := S_OK;
	// ...
	
END_IF	

WritePropertyLogBuffer := _hResult;
END_METHOD

METHOD WritePropertyNotifyType : HRESULT
VAR CONSTANT
	ePropID : E_BACnetPropIdentifier := E_BACnetPropIdentifier.PropNotifyType;
END_VAR
VAR_INPUT
	value : E_BACnet_NotifyType;
END_VAR
IF (ipObj <> 0) THEN
	WritePropertyNotifyType := WriteProperty(ePropID, ADR(value), SIZEOF(value));
ELSE
	WritePropertyNotifyType := E_FAIL;
END_IF
END_METHOD

METHOD WritePropertyNull : HRESULT
VAR_INPUT
	ePropID : E_BACnetPropIdentifier;
	prio : BYTE := 0;
END_VAR
IF (ipObj <> 0) THEN
	WritePropertyNull := ipObj.SyncWriteProperty(TO_INT(ePropID), 0, 0, prio);
	
	IF (WritePropertyNull <> S_OK) THEN
		F_BA_LogMessage2(ADSLOG_MSGTYPE_ERROR, 'WPN5', 'Writing property "%d" failed (Error "0x%x")!', F_INT(ePropID), F_DINT(WritePropertyNull));
	END_IF
ELSE
	WritePropertyNull := E_FAIL;
END_IF
END_METHOD

METHOD WritePropertyReal : HRESULT
VAR_INPUT
	ePropID : E_BACnetPropIdentifier;
	fValue : REAL;
END_VAR
IF (ipObj <> 0) THEN
	WritePropertyReal := WriteProperty(ePropID, ADR(fValue), SIZEOF(fValue));
ELSE
	WritePropertyReal := E_FAIL;
END_IF
END_METHOD

METHOD WritePropertyRealPrio : HRESULT
VAR_INPUT
	ePropID : E_BACnetPropIdentifier;
	fValue : REAL;
	prio : BYTE := 0;
END_VAR
IF (ipObj <> 0) THEN
	WritePropertyRealPrio := ipObj.SyncWriteProperty(TO_INT(ePropID), ADR(fValue), SIZEOF(fValue), prio);
	
	IF (WritePropertyRealPrio <> S_OK) THEN
		F_BA_LogMessage2(ADSLOG_MSGTYPE_ERROR, 'WPRP5', 'Writing property "%d" failed (Error "0x%x")!', F_INT(ePropID), F_DINT(WritePropertyRealPrio));
	END_IF
ELSE
	WritePropertyRealPrio := E_FAIL;
END_IF
END_METHOD

METHOD WritePropertyRecipientList : HRESULT
VAR_IN_OUT
	stRecipientList			: ARRAY[*] OF ST_BACnet_Destination;
END_VAR
// [Bugworkaround]
// > _stUnused" has to be static, otherwise its memory can be initialized incorrectly by PLC :(
VAR_STAT
	_nLowerBound			: DINT;
	_nCount					: DINT;
	_stUnused				: ST_BACnet_Destination;
END_VAR
_hResult := E_FAIL;

IF (ipObj <> 0) THEN
	_nLowerBound := LOWER_BOUND(stRecipientList, 1);
	_nCount := F_BA_GetUsedEntryCount(stRecipientList, _nLowerBound, UPPER_BOUND(stRecipientList, 1), _stUnused);
	
	IF (_nCount > 0) THEN
		_hResult := WriteProperty(E_BACnetPropIdentifier.PropRecipientList, stRecipientList, SIZEOF(ST_BACnet_Destination) * (_nLowerBound + _nCount - 1));
	ELSE
		IF RemoveArrayElements(E_BACnetPropIdentifier.PropRecipientList) THEN
			_hResult := S_OK;
		END_IF
	END_IF
END_IF

WritePropertyRecipientList := _hResult;
END_METHOD

METHOD WritePropertyReference : HRESULT
VAR_INPUT
	eProperty				: E_BACnetPropIdentifier;
END_VAR
VAR_IN_OUT
	stRefObject				: ST_BACnet_ObjectPropertyReference;
END_VAR
VAR
	stTemp					: ST_BACnet_DeviceObjectPropertyReference;
END_VAR
IF (ipObj <> 0) THEN
	IF (stRefObject.iObject = 0) THEN
		// Set referred object to NULL.
	ELSE
		stTemp.stValidFields.bPropertyIdentifier := TRUE;
		stTemp.stValidFields.bObjectId := TRUE;
		
		stTemp.tObjId := stRefObject.iObject.ObjectID;
		stTemp.ePropIdentifier := stRefObject.ePropertyId;
	END_IF
	
	WritePropertyReference := WriteProperty(eProperty, ADR(stTemp), SIZEOF(stTemp));
ELSE
	WritePropertyReference := E_FAIL;
END_IF
END_METHOD

METHOD WritePropertyString : HRESULT
VAR_INPUT
	ePropID : E_BACnetPropIdentifier;
	value : T_MaxString;
END_VAR
VAR
	_nResult : UDINT;
END_VAR
IF (ipObj <> 0) THEN
	IF (F_BACnet_EncodeUTF8(
		pString		:= ADR(value),
		nString	:= TO_UDINT(LEN(value)),
		pResult		:= ADR(BACnet_Globals.stADSBuffer),
		nResult	:= SIZEOF(BACnet_Globals.stADSBuffer),
		nResultLen	:= _nResult) <> 0)
			THEN
				WritePropertyString := WriteProperty(ePropID, ADR(BACnet_Globals.stADSBuffer), TO_UINT(_nResult));
	END_IF
END_IF
END_METHOD

METHOD WritePropertyStringIdx : HRESULT
VAR_INPUT
	ePropID : E_BACnetPropIdentifier;
	str : STRING;
	idx : BYTE;
END_VAR
VAR
	_nResult : UDINT;
END_VAR
IF (ipObj <> 0) THEN
	IF (F_BACnet_EncodeUTF8(
		pString		:= ADR(str),
		nString	:= TO_UDINT(LEN(str)),
		pResult		:= ADR(BACnet_Globals.stADSBuffer),
		nResult	:= SIZEOF(BACnet_Globals.stADSBuffer),
		nResultLen	:= _nResult) <> 0)
			THEN
			WritePropertyStringIdx := ipObj.SyncWriteProperty(TO_INT(ePropID), ADR(BACnet_Globals.stADSBuffer),  TO_UINT(F_BACnet_AlignedSize(_nResult)), idx);
			
			IF (WritePropertyStringIdx <> S_OK) THEN
				F_BA_LogMessage2(ADSLOG_MSGTYPE_ERROR, 'WPSI512', 'Writing property "%d" failed (Error "0x%x")!', F_INT(ePropID), F_DINT(WritePropertyStringIdx));
			END_IF
	END_IF
END_IF
END_METHOD

METHOD WritePropertyUDInt : HRESULT
VAR_INPUT
	ePropID : E_BACnetPropIdentifier;
	nValue : UDINT;
END_VAR
IF (ipObj <> 0) THEN
	WritePropertyUDInt := WriteProperty(ePropID, ADR(nValue), SIZEOF(nValue));
ELSE
	WritePropertyUDInt := E_FAIL;
END_IF
END_METHOD

METHOD WritePropertyUInt : HRESULT
VAR_INPUT
	ePropID : E_BACnetPropIdentifier;
	nValue : UINT;
END_VAR
IF (ipObj <> 0) THEN
	WritePropertyUInt := WriteProperty(ePropID, ADR(nValue), SIZEOF(nValue));
ELSE
	WritePropertyUInt := E_FAIL;
END_IF
END_METHOD

METHOD WritePropertyUnit : HRESULT
VAR CONSTANT
	ePropID : E_BACnetPropIdentifier := E_BACnetPropIdentifier.PropUnits;
END_VAR
VAR_INPUT
	eValue : E_BA_Unit;
END_VAR
IF (ipObj <> 0) THEN
	WritePropertyUnit := WriteProperty(ePropID, ADR(eValue), SIZEOF(eValue));
ELSE
	WritePropertyUnit := E_FAIL;
END_IF
END_METHOD

METHOD WritePropertyValue : HRESULT
VAR_INPUT
	eProperty : E_BACnetPropIdentifier;
	xValue : ANY;
END_VAR
VAR
	_eValueChoice : E_BACnet_ValueChoice;
END_VAR
CASE (xValue.TypeClass) OF
	__SYSTEM.TYPE_CLASS.TYPE_REAL:
		_eValueChoice := E_BACnet_ValueChoice.eRealValue;
	__SYSTEM.TYPE_CLASS.TYPE_UDINT:
		_eValueChoice := E_BACnet_ValueChoice.eUnsignedValue;
	__SYSTEM.TYPE_CLASS.TYPE_BOOL:
		_eValueChoice := E_BACnet_ValueChoice.eBoolValue;
	__SYSTEM.TYPE_CLASS.TYPE_ENUM:
		_eValueChoice := E_BACnet_ValueChoice.eEnumerationValue;
ELSE
	iOwner.LogMsg.Show1(ADSLOG_MSGTYPE_ERROR, 'WPV30', 'Unimplemented datatype! (Type class "%d")', F_DWORD(xValue.TypeClass), TRUE);
	RETURN;
END_CASE

WritePropertyValue := WritePropertyValueEx(eProperty, _eValueChoice, xValue.diSize, xValue.pValue);
END_METHOD

METHOD WritePropertyValueEx : HRESULT
VAR_INPUT
	eProperty : E_BACnetPropIdentifier;
	eValueChoice : E_BACnet_ValueChoice;
	nSize : DINT;
	pValue : PVOID;
END_VAR
VAR
	_stData : ST_BACnet_ValueList;
	_nSize : DWORD;
END_VAR
IF (bReady) AND (nSize > 0) AND (pValue <> 0) THEN
	IF (eValueChoice = E_BACnet_ValueChoice.eEnumerationValue) THEN
		_nSize := SIZEOF(ST_BACnet_ValueList);	
		_stData.nEntrySize := TO_DWORD(SIZEOF(ST_BACnet_Value));
		_stData.listEntry.eValueChoice := eValueChoice;
		_stData.listEntry.nSize := SIZEOF(ST_BACnet_EnumerationValueType);
		_stData.listEntry.stValue.choice := E_BACnet_EnumerationValueChoice.eBinaryPV;
		_stData.listEntry.stValue.enumValue := 0;
		
		MEMCPY(ADR(_stData.listEntry.stValue.enumValue), pValue, TO_UDINT(nSize)); 
	ELSE		
		_nSize := ((SIZEOF(ST_BACnet_ValueList) - SIZEOF(ST_BACnet_EnumerationValueType)) + TO_DWORD(nSize));
		
		_stData.nEntrySize := TO_DWORD((SIZEOF(ST_BACnet_Value) - SIZEOF(ST_BACnet_EnumerationValueType) + nSize));
		_stData.listEntry.eValueChoice := eValueChoice;
		_stData.listEntry.nSize := TO_DWORD(nSize);
		
		MEMCPY(ADR(_stData.listEntry.stValue), pValue, TO_UDINT(nSize)); 
	END_IF
	
	WritePropertyValueEx := WriteProperty(eProperty, ADR(_stData), TO_DINT(F_BACnet_AlignedSize(_nSize)));
				
	IF (S_OK <> WritePropertyValueEx) THEN
		iOwner.LogMsg.Show1(ADSLOG_MSGTYPE_ERROR, 'WPVE12', 'Writing value of property "%d" failed!', F_INT(eProperty), TRUE);
	END_IF
END_IF
END_METHOD

METHOD WritePropertyWeeklySched : HRESULT
VAR_IN_OUT
	stWeek							: ARRAY[*, *] OF ST_BA_SchedEntry;
END_VAR
VAR_INPUT
	eValueChoice					: E_BACnet_ValueChoice;
END_VAR
VAR
	_cbTmpSize						: UDINT;
	_cbTotalEntry					: UDINT;
	_cbTotalBuf						: UDINT;
	_pDailySched					: POINTER TO ST_BACnet_DailySchedule;
	_pTimeValue						: POINTER TO ST_BACnet_TimeValueList;
	_pOldTimeValue					: POINTER TO ST_BACnet_TimeValueList;
	_nDayTmp						: DINT;
	_nDayEntryTmp					: DINT;
	_nDays							: UINT;
END_VAR
IF (ipObj = 0) THEN
	_hResult := E_FAIL;
ELSE
	// Point to first data:
	_pDailySched := ADR(BACnet_Globals.bDefaultBuffer);
	_cbTotalBuf := 0;
	_nDayTmp := LOWER_BOUND(stWeek, 1);
	_hResult := S_OK;
	
	WHILE SUCCEEDED(_hResult) DO
		// Set timevalue pointer:
		_pTimeValue := ADR(_pDailySched^.stListEntry);
		_pTimeValue^.nEntrySize := 0;
		_pTimeValue^.nRes := 0;
		_cbTotalEntry := 0;
		_pOldTimeValue := 0;
		
		FOR _nDayEntryTmp := LOWER_BOUND(stWeek, 2) TO UPPER_BOUND(stWeek, 2) DO
			IF (stWeek[_nDayTmp, _nDayEntryTmp].eState = E_BA_SchedEntryState.eValue) THEN
				// Set flag "next entry" to the previous element:
				IF (_nDayEntryTmp > 1) AND (_pOldTimeValue <> 0) THEN
					_pOldTimeValue^.nEntrySize := _pOldTimeValue^.nEntrySize + 16#80000000;
				END_IF
				
				Sched_WriteEntry(eValueChoice, _pTimeValue, stWeek[_nDayTmp, _nDayEntryTmp]); 
				
				// Update time value pointer:
				Sched_SetNextTimeVal(_pDailySched, _pTimeValue, _cbTmpSize, _pOldTimeValue);
				
				// ...and add to total entry size counter:
				_cbTotalEntry := _cbTotalEntry + _cbTmpSize;
			END_IF
		END_FOR
		
		// Caclulate day-entry size:
		_pDailySched^.nEntrySize := MAX(_cbTotalEntry, SIZEOF(_pDailySched^.stListEntry.nEntrySize) + SIZEOF(_pDailySched^.stListEntry.nRes));
		
		// Next day?
		IF (_nDayTmp < UPPER_BOUND(stWeek, 1)) THEN
			_pDailySched^.nEntrySize := _pDailySched^.nEntrySize + 16#80000000;
		END_IF
		
		// Update pointer each cycle (even if no day follows!):
		IF NOT Sched_SetNextDay(_pDailySched, _cbTmpSize, _cbTotalBuf, _pOldTimeValue, _nDayTmp, _nDayEntryTmp, _pTimeValue) THEN
			EXIT;
		END_IF
	END_WHILE
	
	// Write data:
	_hResult := WriteProperty(E_BACnetPropIdentifier.PropWeeklySchedule, ADR(BACnet_Globals.bDefaultBuffer), TO_DINT(_cbTotalBuf));
END_IF	

WritePropertyWeeklySched := _hResult;
END_METHOD

END_FUNCTION_BLOCK

// POUs/Local/FB_BACnet_Server
FUNCTION_BLOCK FB_BACnet_Server
VAR_INPUT CONSTANT
	{region 'Fixed Parameters'}
		{attribute 'parameterCategory':='General'}
		Adapter	: REFERENCE TO FB_BACnet_Adapter := BACnet_Globals.DefaultAdapter;
	{endregion}
END_VAR
VAR_INPUT CONSTANT PERSISTENT
	{region 'Variable Parameters'}
		{attribute 'parameterCategory':='General'}
		bSupportBackup : BOOL;							// Support backup of PLC persistent data when BACnet backup service is used
		{attribute 'parameterCategory':='General'}
		bDisableWOC : BOOL;								// Deactivate write-on-change mechanism
		{attribute 'parameterCategory':='General'}
		tAmsPort : T_AmsPort := 1000;					// Default port when port can not be determined automatically
	{endregion}
END_VAR
VAR_INPUT CONSTANT
	{region 'Operational Parameters'}
		{attribute 'parameterCategory':='General'}
		bReset : BOOL;									// Manual trigger to reset errors
		{attribute 'parameterCategory':='General'}
		bWritePersistent : BOOL;						// Manual trigger for PLC and BACnet persistent data storage
		{attribute 'parameterCategory':='General'}
		bReload : BOOL;									// Manual trigger to reload ADS connection and increase reload counter (trigger autoget)
	{endregion}
END_VAR
VAR_OUTPUT
	nRevision				: DINT := -1;					// Protocol revision no.
	stAdsConn				: ST_BACnet_AdsConnection;
	eSystemStatus			: E_BACnet_DeviceStatus;
	bBackupActive			: BOOL;
	bWritePersisActive		: BOOL;
	bOperational			: BOOL;
	bWOCDisabled			: BOOL;
	bFirstCycle				: BOOL;
	bInitialized			: BOOL;
	eErrorID				: E_BACnet_Error;
END_VAR
VAR
	{region 'General'}
		nUpdateCount	 	: UDINT := 0;
		nUpdateCountAdp 	: UDINT := 0;
	{endregion}
	{region 'Object-List'}
		{attribute 'hide'}
		pObjList			: POINTER TO ST_ObjectListEntry;
		nObjListCount		: UDINT;
	{endregion}
	{region 'Interface Pointer'}
		{attribute 'hide'}
		oServerOID			: OTCID; 
		{attribute 'hide'}
		iServer 			: ITcIoBACnetPlcServer;	
		{attribute 'hide'}
		bDeleteUnusedObjs	: BOOL := FALSE;
		{attribute 'hide'}
		iDevice				: ITcIoBACnetPlcDevice;
		{attribute 'hide'}
		oDeviceOID			: OTCID;
		{attribute 'hide'}
		iObject				: ITcIoBACnetPlcObject;
	{endregion}
	{region 'Internal'}
		_ObjectId			: DWORD;	
		_SystemStatus		: WORD;			(* ~(BACnet_ObjectType		:  DEV	: )	*)
		_ServerStatus		: WORD;
		_ServerControl		: WORD;
		_fbWritePersistent	: FB_WritePersistentData;
		_rtrigBackup		: R_TRIG;
		_rtrigReset			: R_TRIG;
	
		_bHasStarted		: BOOL := TRUE;
		_nPlcPort			: T_AmsPort;
	{endregion}
	{region 'Misc'}
		{attribute 'hide'}
		fbLogMsg			: FB_BA_LogMessage;
	{endregion}
	{region 'Temporary'}
		_hResult			: HRESULT;
	{endregion}
END_VAR

(* update adapter *)
IF Adapter._nUpdateCount = nUpdateCountAdp THEN
	Adapter();
END_IF
(* remind current number of update counter *)
nUpdateCountAdp := Adapter._nUpdateCount;

IF iDevice = 0 THEN
	iDevice := Adapter.Device;
	IF iDevice <> 0 THEN
		iDevice.TcAddRef();
	END_IF
END_IF


BackupSTM();

IF NOT Error THEN
	IF iServer = 0 THEN
		IF iDevice <> 0 THEN
			iDevice.GetClientById(16#FFFFFFFF, ADR(iServer));
		ELSIF oServerOID <> 0 THEN
			FW_ObjMgr_GetObjectInstance( oid:=oServerOID, iid:=TC_GLOBAL_IID_LIST.IID_ITcIoBACnetPlcServer, pipUnk:=ADR(iServer) );			
		END_IF
		IF iServer <> 0 THEN
			_hResult := iServer.GetAdsPort(ADR(tAmsPort));
			IF SUCCEEDED(_hResult) THEN
				_hResult := iServer.GetObjectByObjectId(ADR(iObject), 16#23FFFFF);
				IF SUCCEEDED(_hResult) THEN
					_hResult := SEL(ReadPropertyUint(E_BACnetPropIdentifier.PropObjectIdentifier, _ObjectId), E_FAIL, S_OK);
				END_IF
				IF SUCCEEDED(_hResult) THEN
					_hResult := iObject.GetPropertyValue(E_BACnetPropIdentifier.PropProtocolRevision, ADR(nRevision), 0);
				END_IF
				eErrorID := SEL(SUCCEEDED(_hResult), E_BACnet_Error.eInvalidServer, E_BACnet_Error.eNoError);
			END_IF
			_hResult := iServer.OnPlcAction(E_BACnet_PlcAction.eStart);
			IF S_OK <> _hResult THEN // Start up
				eErrorID:=E_BACnet_Error.eInvalidTask;
				FW_SafeRelease(ADR(iServer));
				iServer:=0;
				
				fbLogMsg.Show(ADSLOG_MSGTYPE_ERROR, 'D42', 'Task configuration invalid!', FALSE);
			ELSIF iDevice = 0 THEN
				oDeviceOID := iServer.GetBACnetDeviceOid();
				IF oDeviceOID <> 0 THEN
					FW_ObjMgr_GetObjectInstance( oid:=oDeviceOID, iid:=TC_GLOBAL_IID_LIST.IID_ITcIoBACnetPlcDevice, pipUnk:=ADR(iDevice) );
				END_IF
			END_IF
			bDeleteUnusedObjs:=TRUE;
		END_IF
	ELSE
		IF bDeleteUnusedObjs THEN
			_hResult := iServer.OnPlcAction(E_BACnet_PlcAction.eCreateFinish);
			IF S_OK = _hResult THEN
				bDeleteUnusedObjs:=FALSE;
			END_IF
		END_IF	
	END_IF
END_IF

eSystemStatus := E_BACnet_DeviceStatus.Invalid;
IF iDevice <> 0 THEN
	iDevice.GetDeviceStatus(ADR(_SystemStatus));
	eSystemStatus := TO_INT(_SystemStatus);
END_IF

(* control *)
(* Disable write-on-change *)
_ServerControl.2	:= bDisableWOC;
(* PLC running - process data valid *)
_ServerControl.11	:=	(NOT _bHasStarted) AND bOperational;

// Update state:
IF iServer <> 0 THEN
	iServer.UpdateDeviceStatus(ADR(_ServerControl), ADR(_ServerStatus));
	bInitialized := TRUE;
END_IF

(* state *)
//bWritePersisActive := (_iPersis > 0) AND (_iPersis < 100);			// (BETA) ... Trigger Write persistent
bBackupActive := (eSystemStatus = E_BACnet_DeviceStatus.eBackupInProgress);
bOperational :=	SEL(IsValid, FALSE, (Adapter.eAdapterStatus > E_BACnet_AdapterStatus.eInit));
bWOCDisabled := (_ServerStatus AND 16#0004) = 16#0004;

bFirstCycle := (nUpdateCount = 0) AND _bHasStarted;

IF (bFirstCycle) THEN
	// Validate user settings:
	IF (NOT F_BACnet_IsSchedBTypeValid(BACnet_Param.eSched_BType)) THEN
		fbLogMsg.Show(ADSLOG_MSGTYPE_ERROR, 'S90', 'Global parameter "eSchedB_Type" is invalid!', FALSE);
	END_IF
	
ELSIF (NOT bOperational) THEN
	IF Error OR bInitialized THEN
		fbLogMsg.Show(ADSLOG_MSGTYPE_ERROR, 'S95', 'Server device is not operational!', FALSE);
	END_IF

END_IF

_bHasStarted := FALSE;
nUpdateCount := (nUpdateCount+1);

{attribute 'hide'}
METHOD GetObject : BOOL
VAR_INPUT
	tObjectID	: T_BACnet_ObjectIdentifier;
END_VAR
VAR_OUTPUT
	iResult		: I_BACnet_Object;
END_VAR
VAR
	_n : UDINT;
END_VAR
FOR _n:=0 TO nObjListCount DO
	IF pObjList[_n].tObjectID = tObjectID THEN
		iResult:=pObjList[_n].pObject;
		GetObject := (iResult<>0);
		RETURN;
	END_IF
END_FOR
END_METHOD

{attribute 'hide'}
METHOD RegisterObject : BOOL
VAR_INPUT
	tObjectID : T_BACnet_ObjectIdentifier;
	iObject	  : I_BACnet_Object;
END_VAR
VAR
	pTmpTable : POINTER TO ST_ObjectListEntry := 0;
	nTmp : UDINT;
END_VAR
IF F_BACnet_IsObjIdentifierValid(tObjectID) AND (iObject <> 0) THEN
	IF nObjListCount MOD 1000 = 0 THEN
		// Expand list:
		IF pObjList <> 0 THEN
			pTmpTable := pObjList;
			__DELETE(pObjList);
		END_IF
		nTmp := SIZEOF(ST_ObjectListEntry) * (nObjListCount+1000);
		pObjList := __NEW(BYTE, nTmp);
		IF pObjList = 0 THEN
			RETURN;
		END_IF
		IF pTmpTable <> 0 THEN
			MEMCPY(pObjList, pTmpTable, SIZEOF(ST_ObjectListEntry)*nObjListCount);
		END_IF
	END_IF
	
	// Register object:
	pObjList[nObjListCount].pObject := iObject;
	pObjList[nObjListCount].tObjectID := tObjectID;
	nObjListCount := (nObjListCount+1);
	
	RegisterObject := TRUE;
END_IF
END_METHOD

{attribute 'hide'}
PROPERTY ObjectCount : UDINT
GET
VAR
	cnt : UDINT;
END_VAR
IF iObject = 0 THEN
	ObjectCount:=0;
	RETURN;
END_IF

IF S_OK = iObject.SyncReadProperty(E_BACnetPropIdentifier.PropObjectList, ADR(cnt), 0, 0) THEN
 	ObjectCount:=cnt;
	RETURN;
END_IF

ObjectCount:=0;
END_GET
END_PROPERTY

{attribute 'hide'}
PROPERTY ServerItf : ITcIoBACnetPlcServer
GET
ServerItf := iServer;
END_GET
END_PROPERTY

METHOD PRIVATE BackupSTM : BOOL
VAR_INPUT
END_VAR
(* reset trigger *)
_rtrigReset(CLK:= bReset, Q=> );
(* reset error ID and flag *)
IF (eErrorID < 20) OR (eErrorID >= 30) OR _rtrigReset.Q THEN
	eErrorID := E_BACnet_Error.eNoError;
END_IF

(* check if NetID is plausible *)
IF Adapter.sAmsNetId = '' THEN
	(* NetId not OK, return with error *)
	eErrorID := E_BACnet_Error.eNoValidNetId;
END_IF



// (BETA) ... Trigger Write persistent
//IF ((bSupportBackup) OR (_fbWritePersistent.START AND (_iPersis = 0))) THEN
//	(* PLC can be backup't *)
//	_ServerControl.0 := TRUE;
//ELSE
//	(* don't support PLC backup *)
//	_ServerControl.0 := FALSE;
//	_ServerControl.1 := FALSE;
//END_IF




// (BETA) ... Trigger Write persistent
//(* trigger backup flag *)
//_rtrigBackup(CLK:= (eSystemStatus = eBackupInProgress) AND (_iPersis = 0), Q=> );
//IF (_iPersis = 0) THEN
//	(* only backup if persistent state machine is idle *)
//	IF _rtrigBackup.Q AND _ServerControl.0 THEN
//		(* trigger backup function *)
//		_fbWritePersistent.START := TRUE;
//	ELSIF _fbWritePersistent.START AND (NOT _fbWritePersistent.BUSY) THEN
//		IF _fbWritePersistent.ERR THEN
//			(* backup aborted *)
//			eErrorID := E_BACnet_Error.ePERSISTENT_PLC_WRITE;
//		ELSE
//			(* backup was successful *)
//			_ServerControl.1 := TRUE;
//		END_IF
//	ELSIF (eSystemStatus <> eBackupInProgress) THEN
//		(* backup process finished *)
//		_ServerControl.1 := FALSE;
//	END_IF
//END_IF





(* calculate PLC runtime port *)
_nPlcPort := TwinCAT_SystemInfoVarList._AppInfo.AdsPort;

(* call persistent backup *)
(*
_fbWritePersistent(
	NETID	:= '',
	PORT	:= _nPlcPort,
	START	:= ,
	TMOUT	:= BACnet_PlcPersisTimeOut,			// <-- War in BACnet_Param:		BACnet_PlcPersisTimeOut : TIME := T#2M;
	MODE	:= SPDM_VAR_BOOST,
	BUSY	=> ,
	ERR		=> ,
	ERRID	=>
);
*)
END_METHOD

METHOD PRIVATE Reset
IF iServer <> 0 THEN
	iServer.OnPlcAction(E_BACnet_PlcAction.eSuspend); // SUSPEND - delete all pointers to PLC
	FW_SafeRelease(ADR(iServer));
	iServer:=0;
END_IF
IF iObject <> 0 THEN
	FW_SafeRelease(ADR(iObject));
	iObject:=0;
END_IF	
IF iDevice <> 0 THEN
	FW_SafeRelease(ADR(iDevice));
	iDevice:=0;
END_IF 

IF pObjList <> 0 THEN
	__DELETE(pObjList);
	nObjListCount:=0;
END_IF
nObjListCount := 0;

bInitialized := FALSE;
END_METHOD

// Called after online change.
{attribute 'call_after_online_change_slot' := '10'}
METHOD PROTECTED OnPostOnlineChange
Reset();
END_METHOD

METHOD FB_Exit : BOOL
VAR_INPUT
	 bInCopyCode : BOOL; // if TRUE, the exit method is called for exiting an instance that is copied afterwards (online change).
END_VAR
Reset();
END_METHOD

PROPERTY Error : BOOL
GET
Error := (eErrorID <> E_BACnet_Error.eNoError);
END_GET
END_PROPERTY

PROPERTY IsValid : BOOL
GET
IsValid := (_ObjectId <> 16#00000000);
END_GET
END_PROPERTY

{attribute 'hide'}
METHOD ReadPropertyUint : BOOL
VAR_INPUT
	ePropID : E_BACnetPropIdentifier;
	value : REFERENCE TO UDINT;
END_VAR
VAR
	_hr : HRESULT;
	_size : DINT := 4;
END_VAR
IF iObject<>0 AND (__ISVALIDREF(value)) THEN
	_hr:=iObject.SyncReadProperty(TO_INT(ePropID), ADR(value), ADR(_size), 16#FFFFFFFF);
	IF (_hr = S_OK) THEN
		ReadPropertyUint:=TRUE;
		RETURN;
	END_IF
END_IF
ReadPropertyUint:=FALSE;
END_METHOD

END_FUNCTION_BLOCK

// POUs/FB_BACnet_Adapter
FUNCTION_BLOCK FB_BACnet_Adapter
VAR_OUTPUT
	eAdapterStatus				: E_BACnet_AdapterStatus;
	bEthernetLink				: BOOL;
	bGateway					: BOOL;
	sAmsNetId					: T_AmsNetId;
	bFirstCycle					: BOOL;
	eErrorID					: E_BACnet_Error;
END_VAR
VAR
	BACnet_AmsNetId		AT %I*	: ARRAY[0 .. 5] OF BYTE;	(* ~(BACnet_AmsNetId : : ) *)
	
	_DeviceStatus				: WORD;
	_bHasStarted				: BOOL						:= TRUE;
	_nUpdateCount				: UDINT						:= 0;
	iDevice						: ITcIoBACnetPlcDevice;
	_fbAdsRead					: FW_AdsRead;
    oAdapterOID  				: OTCID;
	
	{attribute 'hide'}
	fbLogMsg					: FB_BA_LogMessage;
	
	_hResult					: HRESULT;
END_VAR
VAR_STAT
	// (BETA) ... Following symbols should be made non-static / thread safe!
	{region 'Temporary'}
		{attribute 'hide'}
		_bErrTmp					: BOOL;
	{endregion}
END_VAR

// Reset error ID
eErrorID := E_BACnet_Error.eNoError;

IF iDevice = 0 THEN
	IF oAdapterOID = 0 THEN
		IF sAmsNetId = '' THEN
			// Read NetId and convert to string:
			sAmsNetId := F_CreateAmsNetId(BACnet_AmsNetId);
			
			// Check if it plausible:
			IF sAmsNetId = BACnet_Globals.tInvalidAmsNetId THEN
				eErrorID := E_BACnet_Error.eNoValidNetId;
				
				F_BA_LogMessage(ADSLOG_MSGTYPE_ERROR, 'UNID06', 'BACnet Adapter: AmsNet-ID is not linked to respective device!');
			END_IF
		ELSE
			eErrorID := E_BACnet_Error.eNoValidNetId;
		END_IF
		
		// Check if it plausible:
		IF sAmsNetId <> BACnet_Globals.tInvalidAmsNetId THEN
			_fbAdsRead(
				sNetId		:= sAmsNetId,
				nPort		:= 16#FFFF,
				nIdxGrp		:= 16#80000033,
				nIdxOffs	:= 0,
				cbReadLen	:= SIZEOF(oAdapterOID),
				pReadBuff	:= ADR(oAdapterOID),
				bExecute	:= TRUE,
				tTimeout	:= BACnet_Param.tADS_TimeOut,
				bBusy		=> ,
				bError		=> _bErrTmp,
				nErrId		=> ,
				cbRead		=> );
				
			IF (_bErrTmp) THEN
				eErrorID := E_BACnet_Error.eADS_NoValidNetId;
			END_IF
		END_IF
	END_IF
	IF oAdapterOID <> 0 THEN
		IF S_OK <> FW_ObjMgr_GetObjectInstance( oid:=oAdapterOID, iid:=TC_GLOBAL_IID_LIST.IID_ITcIoBACnetPlcDevice, pipUnk:=ADR(iDevice) ) THEN
			eErrorID := E_BACnet_Error.eDeviceNotFound;
		END_IF
	END_IF
ELSE
	_hResult := iDevice.CycleTask();
	IF S_OK <> _hResult THEN
		eErrorID := E_BACnet_Error.eInvalidTask;
		fbLogMsg.Show(ADSLOG_MSGTYPE_ERROR, 'D63', 'Task configuration invalid!', FALSE);
	END_IF			
END_IF

IF iDevice <> 0 THEN
	iDevice.GetDeviceStatus(ADR(_DeviceStatus));
	// Convert _DeviceStatus to enumeration
	eAdapterStatus := TO_INT(SHR((_DeviceStatus AND 16#FF00), 8));
	// States
	bEthernetLink := (NOT _DeviceStatus.0);
	bGateway := (eAdapterStatus = E_BACnet_AdapterStatus.eComplete) AND bEthernetLink;
END_IF

// Update counter
IF (_nUpdateCount = 0) AND _bHasStarted THEN
	bFirstCycle := TRUE;
	_bHasStarted := FALSE;
ELSE
	bFirstCycle := FALSE;
END_IF
_nUpdateCount := (_nUpdateCount+1);

METHOD FB_exit : BOOL
VAR_INPUT
	 bInCopyCode : BOOL; // if TRUE, the exit method is called for exiting an instance that is copied afterwards (online change).
END_VAR
IF oAdapterOID <> 0 THEN
	IF iDevice <> 0 THEN
		FW_SafeRelease(ADR(iDevice));
		iDevice:=0;
	END_IF
END_IF
END_METHOD

METHOD FB_init : BOOL
VAR_INPUT
	bInitRetains : BOOL; // if TRUE, the retain variables are initialized (warm start / cold start)
	bInCopyCode : BOOL;  // if TRUE, the instance afterwards gets moved into the copy code (online change)
END_VAR
END_METHOD

METHOD GetDiagnosis : BOOL
VAR_INPUT
	pDiag : POINTER TO ST_BACnet_Diagnosis;
END_VAR
IF iDevice <> 0 THEN
	IF S_OK = iDevice.GetDeviceData(pDiag, SIZEOF(ST_BACnet_Diagnosis), 1) THEN
		GetDiagnosis:=TRUE;
	END_IF
END_IF
END_METHOD

METHOD ResetDiagnosis : BOOL
VAR_INPUT
END_VAR
IF iDevice <> 0 THEN
	IF S_OK = iDevice.GetDeviceData(0, 0, 16#80000001) THEN
		ResetDiagnosis:=TRUE;
	END_IF
END_IF
END_METHOD

PROPERTY Device :  ITcIoBACnetPlcDevice
GET
Device := iDevice;
END_GET
SET
iDevice := Device;
END_SET
END_PROPERTY

PROPERTY Error : BOOL
GET
Error := (eErrorID <> E_BACnet_Error.eNoError);
END_GET
END_PROPERTY

METHOD GetScanResult : BOOL
VAR_INPUT
	pScanRes : POINTER TO ST_BACnetRM_ScanResult;
	nScanResMaxEntries : UDINT;
END_VAR
IF iDevice <> 0 THEN
	IF S_OK = iDevice.GetDeviceData(pScanRes, SIZEOF(ST_BACnetRM_ScanResult)*nScanResMaxEntries, 16#00000002) THEN
		GetScanResult:=TRUE;
	END_IF
END_IF
END_METHOD

METHOD StartScan : BOOL
VAR_INPUT
END_VAR
IF iDevice <> 0 THEN
	IF S_OK = iDevice.StartScan(0,0) THEN
		StartScan:=TRUE;
	END_IF
END_IF
END_METHOD

METHOD StartScanEx : BOOL
VAR_INPUT
	bRescrictID	 : BOOL;
	bRestrictNet : BOOL;
	bLocalBroadcast : BOOL;
	nNetNr : UINT;
	nStartID : UDINT;
	nEndID : UDINT;
END_VAR
VAR
	scanRes : ST_BACnetRM_ScanParameter;
END_VAR
IF iDevice <> 0 THEN
	scanRes.bRescrictID:=bRescrictID;
	scanRes.bRestrictNet:=bRestrictNet;
	scanRes.bLocalBroadcast:=bLocalBroadcast;
	scanRes.nNetNr:=nNetNr;
	scanRes.nStartID:=nStartID;
	scanRes.nEndID:=nEndID;
	IF S_OK = iDevice.StartScan(ADR(scanRes),SIZEOF(ST_BACnetRM_ScanParameter)) THEN
		StartScanEx:=TRUE;
	END_IF
END_IF
END_METHOD

METHOD TimeSync : BOOL
VAR_INPUT
	pDateTime : POINTER TO ST_BA_DateTime;
	bSendBroadcast : BOOL;
END_VAR
IF iDevice <> 0 THEN
	IF S_OK = iDevice.TimeSync(pDateTime, NOT bSendBroadcast) THEN
		TimeSync:=TRUE;
	END_IF
END_IF
END_METHOD

END_FUNCTION_BLOCK

// POUs/Local/Objects/FB_BACnet_View
// Structured View Object
FUNCTION_BLOCK FB_BACnet_View EXTENDS FB_BACnet_Object IMPLEMENTS I_BACnet_View
VAR_INPUT CONSTANT
	{attribute 'parameterCategory':='General'}
	eNodeType : E_BACnet_NodeType := E_BACnet_NodeType.eOrganizational;
END_VAR

SUPER^();

METHOD PROTECTED OnObjectStateChanged
SUPER^.OnObjectStateChanged();

CASE (tState) OF
	TCOM_STATE.TCOM_STATE_PREOP:
		// SyncHandler:
		RequestSyncHandlers(0, 1);
		
	TCOM_STATE.TCOM_STATE_SAFEOP:
		;

	TCOM_STATE.TCOM_STATE_OP:
		SyncProperty(E_BACnetPropIdentifier.PropNodeType, SIZEOF(eNodeType), ADR(eNodeType), 0, eFullSync_InitPLC, FALSE);
		
END_CASE
END_METHOD

METHOD FB_init : BOOL
VAR_INPUT
	bInitRetains : BOOL; // if TRUE, the retain variables are initialized (warm start / cold start)
	bInCopyCode : BOOL;  // if TRUE, the instance afterwards gets moved into the copy code (online change)
END_VAR
eObjectType := E_BACnetObjType.ObjStructuredView;
END_METHOD

END_FUNCTION_BLOCK

// POUs/Local/Objects/[Base]/FB_BACnet_BaseAI
FUNCTION_BLOCK FB_BACnet_BaseAI EXTENDS FB_BACnet_EventObject
VAR_INPUT CONSTANT PERSISTENT
	{region 'Variable Parameters'}
		{attribute 'parameterCategory':='Hardware'}
		{attribute 'TcEncoding':='UTF-8'}
		sDeviceType : STRING;
		{attribute 'parameterCategory':='Hardware'}
		{attribute 'parameterUnit':= '1/100s'}
		nUpdateInterval : UDINT := 5;
		
		{attribute 'parameterCategory':='Value'}
		fMinPresValue : REAL := 0;
		{attribute 'parameterCategory':='Value'}
		fMaxPresValue : REAL := 100;
		{attribute 'parameterCategory':='Value'}
		fFaultDeadband : REAL := 0.0;
		{attribute 'parameterCategory':='Value'}
		bEnOutOfService : BOOL;
		{attribute 'parameterCategory':='Value'}
		fCOVIncrement : REAL := 0.1;
		{attribute 'parameterCategory':='Value'}
		nAvgFilterCycles : UDINT := 0;
		{attribute 'parameterCategory':='Value'}
		eUnit : E_BA_Unit := E_BA_Unit.eOther_NoUnits;
		
		{attribute 'parameterCategory':='EventConfig'}
		bLowLimitEnable : BOOL := FALSE;
		{attribute 'parameterCategory':='EventConfig'}
		fLowLimitValue : REAL;
		{attribute 'parameterCategory':='EventConfig'}
		bHighLimitEnable : BOOL := FALSE;
		{attribute 'parameterCategory':='EventConfig'}
		fHighLimitValue : REAL;
		{attribute 'parameterCategory':='EventConfig'}
		fDeadband : REAL := 0.0;
	{endregion}
END_VAR
VAR_OUTPUT
	fPresentValue	: REAL;
END_VAR

SUPER^();

METHOD PROTECTED OnObjectStateChanged
SUPER^.OnObjectStateChanged();

CASE (tState) OF
	TCOM_STATE.TCOM_STATE_PREOP:
		// SyncHandler:
		RequestSyncHandlers(0, 14);
		
		// Ensure UTF-8 Encoding:
		F_BA_EnsureUTF8(ADR(sDeviceType), SIZEOF(sDeviceType));
		
	TCOM_STATE.TCOM_STATE_SAFEOP:
		;
		
	TCOM_STATE.TCOM_STATE_OP:
		SyncProperty(E_BACnetPropIdentifier.PropDeviceType, SIZEOF(sDeviceType), ADR(sDeviceType), 0, eFullSync_InitPLC, FALSE);
		SyncProperty(E_BACnetPropIdentifier.PropUpdateInterval, SIZEOF(nUpdateInterval), ADR(nUpdateInterval), 0, eFullSync_InitPLC, FALSE);
		SyncProperty(E_BACnetPropIdentifier.PropUnits, SIZEOF(eUnit), ADR(eUnit), 0, eFullSync_InitPLC, FALSE);
		SyncProperty(E_BACnetPropIdentifier.PropMinPresValue, SIZEOF(fMinPresValue), ADR(fMinPresValue), 0, eFullSync_InitPLC, FALSE);
		SyncProperty(E_BACnetPropIdentifier.PropMaxPresValue, SIZEOF(fMaxPresValue), ADR(fMaxPresValue), 0, eFullSync_InitPLC, FALSE);
		SyncProperty(E_BACnetPropIdentifier.PropFaultDeadband, SIZEOF(fFaultDeadband), ADR(fFaultDeadband), 0, eFullSync_InitPLC, FALSE);
		SyncProperty(E_BACnetPropIdentifier.PropOutOfService, SIZEOF(bEnOutOfService), ADR(bEnOutOfService), 0, eFullSync_InitPLC, FALSE);
		SyncProperty(E_BACnetPropIdentifier.PropCovIncrement, SIZEOF(fCOVIncrement), ADR(fCOVIncrement), 0, eFullSync_InitPLC, FALSE);
		SyncProperty(E_BACnetPropIdentifier.PropAvgFilterCycles, SIZEOF(nAvgFilterCycles), ADR(nAvgFilterCycles), 0, eFullSync_InitPLC, FALSE);
		SyncPropertyIdx(E_BACnetPropIdentifier.PropLimitEnable, SIZEOF(BOOL), ADR(bHighLimitEnable), E_BACnet_LimitEnableBits.eHighLimit, 0, eFullSync_InitPLC, FALSE);	
		SyncPropertyIdx(E_BACnetPropIdentifier.PropLimitEnable, SIZEOF(BOOL), ADR(bLowLimitEnable), E_BACnet_LimitEnableBits.eLowLimit, 0, eFullSync_InitPLC, FALSE);
		SyncProperty(E_BACnetPropIdentifier.PropHighLimit, SIZEOF(fHighLimitValue), ADR(fHighLimitValue), 0, eFullSync_InitPLC, FALSE);
		SyncProperty(E_BACnetPropIdentifier.PropLowLimit, SIZEOF(fLowLimitValue), ADR(fLowLimitValue), 0, eFullSync_InitPLC, FALSE);
		SyncProperty(E_BACnetPropIdentifier.PropDeadband, SIZEOF(fDeadband), ADR(fDeadband), 0, eFullSync_InitPLC, FALSE);
		
END_CASE
END_METHOD

METHOD FB_init : BOOL
VAR_INPUT
	bInitRetains : BOOL; // if TRUE, the retain variables are initialized (warm start / cold start)
	bInCopyCode : BOOL;  // if TRUE, the instance afterwards gets moved into the copy code (online change)
END_VAR
eObjectType := E_BACnetObjType.ObjAnalogInput;
END_METHOD

END_FUNCTION_BLOCK

// POUs/Local/Objects/[Base]/FB_BACnet_BaseAO
FUNCTION_BLOCK FB_BACnet_BaseAO EXTENDS FB_BACnet_EventObject
VAR_INPUT
	bEnPgm					: BOOL;
	fValPgm					: REAL;
END_VAR
VAR_INPUT CONSTANT PERSISTENT
	{region 'Variable Parameters'}
		{attribute 'parameterCategory':='Hardware'}
		{attribute 'TcEncoding':='UTF-8'}
		sDeviceType : STRING;
		{attribute 'parameterCategory':='Hardware'}
		fResolution : REAL := 0.1;
		{attribute 'parameterCategory':='Hardware'}
		fScaleOffset : REAL := 0;
		
		{attribute 'parameterCategory':='Value'}
		fMinPresValue : REAL := 0;
		{attribute 'parameterCategory':='Value'}
		fMaxPresValue : REAL := 100;
		{attribute 'parameterCategory':='Value'}
		fRelinquishDefault : REAL;
		{attribute 'parameterCategory':='Value'}
		bEnOutOfService : BOOL;
		{attribute 'parameterCategory':='Value'}
		fCOVIncrement : REAL := 0.1;
		{attribute 'parameterCategory':='Value'}
		eUnit : E_BA_Unit := E_BA_Unit.eOther_NoUnits;
		
		{attribute 'parameterCategory':='EventConfig'}
		bLowLimitEnable : BOOL := FALSE;
		{attribute 'parameterCategory':='EventConfig'}
		fLowLimitValue : REAL;
		{attribute 'parameterCategory':='EventConfig'}
		bHighLimitEnable : BOOL := FALSE;
		{attribute 'parameterCategory':='EventConfig'}
		fHighLimitValue : REAL;
		{attribute 'parameterCategory':='EventConfig'}
		fDeadband : REAL := 0.0;
	{endregion}
END_VAR
VAR_OUTPUT
	fPresentValue			: REAL;
END_VAR
VAR
	{region 'Internal'}
		_bOverriddenValue	: BOOL;
	{endregion}
END_VAR

SUPER^();

METHOD PROTECTED OnObjectStateChanged
SUPER^.OnObjectStateChanged();

CASE (tState) OF
	TCOM_STATE.TCOM_STATE_PREOP:
		// SyncHandler:
		RequestSyncHandlers(1, 16);
		
		// Ensure UTF-8 Encoding:
		F_BA_EnsureUTF8(ADR(sDeviceType), SIZEOF(sDeviceType));
		
	TCOM_STATE.TCOM_STATE_SAFEOP:
		SyncPropertyPvPrio(E_BACnetPropIdentifier.PropPresentValue, SIZEOF(fValPgm), ADR(fValPgm), ADR(bEnPgm), BACnet_Param.nPrio_Program, 0, eFullSync_InitPLC, TRUE);
		
		SyncProperty(E_BACnetPropIdentifier.PropPresentValue, SIZEOF(fPresentValue), ADR(fPresentValue), 0, eSync_FromSupplement, TRUE);
		
	TCOM_STATE.TCOM_STATE_OP:
		SyncProperty(E_BACnetPropIdentifier.PropResolution, SIZEOF(fResolution), ADR(fResolution), 0, eFullSync_InitPLC, FALSE);
		SyncProperty(E_BACnetPropIdentifier.PropScaleOffset, SIZEOF(fScaleOffset), ADR(fScaleOffset), 0, eFullSync_InitPLC, FALSE);
		SyncProperty(E_BACnetPropIdentifier.PropDeviceType, SIZEOF(sDeviceType), ADR(sDeviceType), 0, eFullSync_InitPLC, FALSE);
		SyncProperty(E_BACnetPropIdentifier.PropUnits, SIZEOF(eUnit), ADR(eUnit), 0, eFullSync_InitPLC, FALSE);
		SyncProperty(E_BACnetPropIdentifier.PropMinPresValue, SIZEOF(fMinPresValue), ADR(fMinPresValue), 0, eFullSync_InitPLC, FALSE);
		SyncProperty(E_BACnetPropIdentifier.PropMaxPresValue, SIZEOF(fMaxPresValue), ADR(fMaxPresValue), 0, eFullSync_InitPLC, FALSE);
		SyncPropertyIdx(E_BACnetPropIdentifier.PropLimitEnable, SIZEOF(BOOL), ADR(bHighLimitEnable), E_BACnet_LimitEnableBits.eHighLimit, 0, eFullSync_InitPLC, FALSE);	
		SyncPropertyIdx(E_BACnetPropIdentifier.PropLimitEnable, SIZEOF(BOOL), ADR(bLowLimitEnable), E_BACnet_LimitEnableBits.eLowLimit, 0, eFullSync_InitPLC, FALSE);
		SyncProperty(E_BACnetPropIdentifier.PropHighLimit, SIZEOF(fHighLimitValue), ADR(fHighLimitValue), 0, eFullSync_InitPLC, FALSE);
		SyncProperty(E_BACnetPropIdentifier.PropLowLimit, SIZEOF(fLowLimitValue), ADR(fLowLimitValue), 0, eFullSync_InitPLC, FALSE);
		SyncProperty(E_BACnetPropIdentifier.PropDeadband, SIZEOF(fDeadband), ADR(fDeadband), 0, eFullSync_InitPLC, FALSE);
		SyncProperty(E_BACnetPropIdentifier.PropRelinquishDefault, SIZEOF(fRelinquishDefault), ADR(fRelinquishDefault), 0, eFullSync_InitPLC, FALSE);
		SyncProperty(E_BACnetPropIdentifier.PropOutOfService, SIZEOF(bEnOutOfService), ADR(bEnOutOfService), 0, eFullSync_InitPLC, FALSE);
		SyncProperty(E_BACnetPropIdentifier.PropCovIncrement, SIZEOF(fCOVIncrement), ADR(fCOVIncrement), 0, eFullSync_InitPLC, FALSE);
		
		SyncProperty(E_BACnetPropIdentifier.PropRawIoStateOverride, SIZEOF(_bOverriddenValue), ADR(_bOverriddenValue), 0, eSync_ToSupplement, FALSE);
		
END_CASE
END_METHOD

METHOD FB_init : BOOL
VAR_INPUT
	bInitRetains : BOOL; // if TRUE, the retain variables are initialized (warm start / cold start)
	bInCopyCode : BOOL;  // if TRUE, the instance afterwards gets moved into the copy code (online change)
END_VAR
eObjectType := E_BACnetObjType.ObjAnalogOutput;
END_METHOD

END_FUNCTION_BLOCK

// POUs/Local/Objects/[Base]/FB_BACnet_BaseBI
FUNCTION_BLOCK FB_BACnet_BaseBI EXTENDS FB_BACnet_EventObject
VAR_INPUT CONSTANT PERSISTENT
	{region 'Variable Parameters'}
		{attribute 'parameterCategory':='Value'}
		bEnOutOfService : BOOL;
		{attribute 'parameterCategory':='Value'}
		{attribute 'TcEncoding':='UTF-8'}
		sInactiveText : T_BACnet_StateText;
		{attribute 'parameterCategory':='Value'}
		{attribute 'TcEncoding':='UTF-8'}
		sActiveText : T_BACnet_StateText;
		
		{attribute 'parameterCategory':='Hardware'}
		{attribute 'TcEncoding':='UTF-8'}
		sDeviceType : STRING;
		
		{attribute 'parameterCategory':='EventConfig'}
		bAlarmValue : BOOL := TRUE;
		
		{attribute 'parameterCategory':='Config'}
		ePolarity : E_BA_Polarity := E_BA_Polarity.eNormal;
			 
		{attribute 'parameterCategory':='StateChange'}
		nChangeOfStateCount : UDINT;
		
		{attribute 'parameterCategory':='ActiveTime'}
		{attribute 'parameterUnit':= 's'}
		nElapsedActiveTime : UDINT;
	{endregion}
END_VAR
VAR_OUTPUT
	bPresentValue			: BOOL;
END_VAR
VAR
	{region 'Output-Properties'}
		{attribute 'parameterCategory':='StateChange'}
		stChangeOfStateTime : ST_BA_DateTime;
		{attribute 'parameterCategory':='StateChange'}
		stTimeOfStateCountReset : ST_BA_DateTime;
		
		{attribute 'parameterCategory':='ActiveTime'}
		stTimeOfActiveTimeReset : ST_BA_DateTime;
	{endregion}
END_VAR

SUPER^();

METHOD PROTECTED OnObjectStateChanged
SUPER^.OnObjectStateChanged();

CASE (tState) OF
	TCOM_STATE.TCOM_STATE_PREOP:
		// SyncHandler:
		RequestSyncHandlers(4, 8);
		
		// Properties:
		IF (BACnet_Param.bStateText_WriteProtect) THEN
			WriteProtectProperty(E_BACnetPropIdentifier.PropActiveText, TRUE);
			WriteProtectProperty(E_BACnetPropIdentifier.PropInactiveText, TRUE);
		END_IF
		
		// Ensure UTF-8 Encoding:
		F_BA_EnsureUTF8(ADR(sDeviceType), SIZEOF(sDeviceType));
		F_BA_EnsureUTF8(ADR(sInactiveText), SIZEOF(sInactiveText));
		F_BA_EnsureUTF8(ADR(sActiveText), SIZEOF(sActiveText));

	TCOM_STATE.TCOM_STATE_SAFEOP:
		SyncProperty(E_BACnetPropIdentifier.PropPresentValue, SIZEOF(bPresentValue), ADR(bPresentValue), 0, eSync_FromSupplement, TRUE);
		
	TCOM_STATE.TCOM_STATE_OP:
		SyncProperty(E_BACnetPropIdentifier.PropAlarmValue, SIZEOF(bAlarmValue), ADR(bAlarmValue), 0, eFullSync_InitPLC, FALSE);
		SyncProperty(E_BACnetPropIdentifier.PropOutOfService, SIZEOF(bEnOutOfService), ADR(bEnOutOfService), 0, eFullSync_InitPLC, FALSE);
		SyncProperty(E_BACnetPropIdentifier.PropActiveText, SIZEOF(sActiveText), ADR(sActiveText), 0, eFullSync_InitPLC, FALSE);	
		SyncProperty(E_BACnetPropIdentifier.PropInactiveText, SIZEOF(sInactiveText), ADR(sInactiveText), 0, eFullSync_InitPLC, FALSE);
		SyncProperty(E_BACnetPropIdentifier.PropPolarity, SIZEOF(ePolarity), ADR(ePolarity), 0, eFullSync_InitPLC, FALSE);
		SyncProperty(E_BACnetPropIdentifier.PropDeviceType, SIZEOF(sDeviceType), ADR(sDeviceType), 0, eFullSync_InitPLC, FALSE);

		SyncProperty(E_BACnetPropIdentifier.PropChangeOfStateCount, SIZEOF(nChangeOfStateCount), ADR(nChangeOfStateCount), 0, eFullSync_InitPLC, FALSE);
		SyncProperty(E_BACnetPropIdentifier.PropChangeOfStateTime, SIZEOF(stChangeOfStateTime), ADR(stChangeOfStateTime), 0, eSync_FromSupplement, FALSE);
		SyncProperty(E_BACnetPropIdentifier.PropTimeOfStateCountReset, SIZEOF(stTimeOfStateCountReset), ADR(stTimeOfStateCountReset), 0, eSync_FromSupplement, FALSE);

		SyncProperty(E_BACnetPropIdentifier.PropElapsedActiveTime, SIZEOF(nElapsedActiveTime), ADR(nElapsedActiveTime), 0, eFullSync_InitPLC, FALSE);
		SyncProperty(E_BACnetPropIdentifier.PropTimeOfActiveTimeReset, SIZEOF(stTimeOfActiveTimeReset), ADR(stTimeOfActiveTimeReset), 0, eSync_FromSupplement, FALSE);
		
END_CASE
END_METHOD

METHOD FB_init : BOOL
VAR_INPUT
	bInitRetains : BOOL; // if TRUE, the retain variables are initialized (warm start / cold start)
	bInCopyCode : BOOL;  // if TRUE, the instance afterwards gets moved into the copy code (online change)
END_VAR
eObjectType := E_BACnetObjType.ObjBinaryInput;
END_METHOD

END_FUNCTION_BLOCK

// POUs/Local/Objects/[Base]/FB_BACnet_BaseBO
FUNCTION_BLOCK FB_BACnet_BaseBO EXTENDS FB_BACnet_EventObject
VAR_INPUT
	bEnPgm			: BOOL;
	bValPgm			: BOOL;
END_VAR
VAR_INPUT CONSTANT PERSISTENT
	{region 'Variable Parameters'}
		{attribute 'parameterCategory':='General'}
		{attribute 'parameterUnit':= 's'}
		nMinimumOffTime : UDINT;
		{attribute 'parameterCategory':='General'}
		{attribute 'parameterUnit':= 's'}
		nMinimumOnTime : UDINT;
		
		{attribute 'parameterCategory':='Value'}
		bRelinquishDefault : BOOL;
		{attribute 'parameterCategory':='Value'}
		bEnOutOfService : BOOL;
		{attribute 'parameterCategory':='Value'}
		{attribute 'TcEncoding':='UTF-8'}
		sInactiveText : T_BACnet_StateText;
		{attribute 'parameterCategory':='Value'}
		{attribute 'TcEncoding':='UTF-8'}
		sActiveText : T_BACnet_StateText;
		
		{attribute 'parameterCategory':='Hardware'}
		{attribute 'TcEncoding':='UTF-8'}
		sDeviceType : STRING;
		
		{attribute 'parameterCategory':='Config'}
		ePolarity : E_BA_Polarity := E_BA_Polarity.eNormal;
			 
		{attribute 'parameterCategory':='StateChange'}
		nChangeOfStateCount : UDINT;
		
		{attribute 'parameterCategory':='ActiveTime'}
		{attribute 'parameterUnit':= 's'}
		nElapsedActiveTime : UDINT;
	{endregion}
END_VAR
VAR_OUTPUT
	bPresentValue	: BOOL;
END_VAR
VAR
	{region 'Output-Properties'}
		{attribute 'parameterCategory':='StateChange'}
		stChangeOfStateTime : ST_BA_DateTime;
		{attribute 'parameterCategory':='StateChange'}
		stTimeOfStateCountReset : ST_BA_DateTime;
		
		{attribute 'parameterCategory':='ActiveTime'}
		stTimeOfActiveTimeReset : ST_BA_DateTime;
	{endregion}
END_VAR
VAR
	{region 'General'}
		_bFeedbackValue	: BOOL;
	{endregion}
END_VAR

SUPER^();

METHOD PROTECTED OnObjectStateChanged
SUPER^.OnObjectStateChanged();

CASE (tState) OF
	TCOM_STATE.TCOM_STATE_PREOP:
		// SyncHandler:
		RequestSyncHandlers(4, 12);
		
		// Properties:
		IF (BACnet_Param.bStateText_WriteProtect) THEN
			WriteProtectProperty(E_BACnetPropIdentifier.PropActiveText, TRUE);
			WriteProtectProperty(E_BACnetPropIdentifier.PropInactiveText, TRUE);
		END_IF
		
		// Ensure UTF-8 Encoding:
		F_BA_EnsureUTF8(ADR(sDeviceType), SIZEOF(sDeviceType));
		F_BA_EnsureUTF8(ADR(sInactiveText), SIZEOF(sInactiveText));
		F_BA_EnsureUTF8(ADR(sActiveText), SIZEOF(sActiveText));

	TCOM_STATE.TCOM_STATE_SAFEOP:
		SyncPropertyPvPrio(E_BACnetPropIdentifier.PropPresentValue, SIZEOF(bValPgm), ADR(bValPgm), ADR(bEnPgm), BACnet_Param.nPrio_Program, 0, eFullSync_InitPLC, TRUE);
		
		SyncProperty(E_BACnetPropIdentifier.PropPresentValue, SIZEOF(bPresentValue), ADR(bPresentValue), 0, eSync_FromSupplement, TRUE);
		
		SyncProperty(E_BACnetPropIdentifier.PropFeedbackValue, SIZEOF(_bFeedbackValue), ADR(_bFeedbackValue), 0, eSync_ToSupplement, TRUE);
		
	TCOM_STATE.TCOM_STATE_OP:
		SyncProperty(E_BACnetPropIdentifier.PropDeviceType, SIZEOF(sDeviceType), ADR(sDeviceType), 0, eFullSync_InitPLC, FALSE);
		SyncProperty(E_BACnetPropIdentifier.PropOutOfService, SIZEOF(bEnOutOfService), ADR(bEnOutOfService), 0, eFullSync_InitPLC, FALSE);
		SyncProperty(E_BACnetPropIdentifier.PropMinimumOffTime, SIZEOF(nMinimumOffTime), ADR(nMinimumOffTime), 0, eFullSync_InitPLC, FALSE);	
		SyncProperty(E_BACnetPropIdentifier.PropMinimumOnTime, SIZEOF(nMinimumOnTime), ADR(nMinimumOnTime), 0, eFullSync_InitPLC, FALSE);	
		SyncProperty(E_BACnetPropIdentifier.PropRelinquishDefault, SIZEOF(bRelinquishDefault), ADR(bRelinquishDefault), 0, eFullSync_InitPLC, FALSE);	
		SyncProperty(E_BACnetPropIdentifier.PropActiveText, SIZEOF(sActiveText), ADR(sActiveText), 0, eFullSync_InitPLC, FALSE);	
		SyncProperty(E_BACnetPropIdentifier.PropInactiveText, SIZEOF(sInactiveText), ADR(sInactiveText), 0, eFullSync_InitPLC, FALSE);
		SyncProperty(E_BACnetPropIdentifier.PropPolarity, SIZEOF(ePolarity), ADR(ePolarity), 0, eFullSync_InitPLC, FALSE);

		SyncProperty(E_BACnetPropIdentifier.PropChangeOfStateCount, SIZEOF(nChangeOfStateCount), ADR(nChangeOfStateCount), 0, eFullSync_InitPLC, FALSE);
		SyncProperty(E_BACnetPropIdentifier.PropChangeOfStateTime, SIZEOF(stChangeOfStateTime), ADR(stChangeOfStateTime), 0, eSync_FromSupplement, FALSE);
		SyncProperty(E_BACnetPropIdentifier.PropTimeOfStateCountReset, SIZEOF(stTimeOfStateCountReset), ADR(stTimeOfStateCountReset), 0, eSync_FromSupplement, FALSE);

		SyncProperty(E_BACnetPropIdentifier.PropElapsedActiveTime, SIZEOF(nElapsedActiveTime), ADR(nElapsedActiveTime), 0, eFullSync_InitPLC, FALSE);
		SyncProperty(E_BACnetPropIdentifier.PropTimeOfActiveTimeReset, SIZEOF(stTimeOfActiveTimeReset), ADR(stTimeOfActiveTimeReset), 0, eSync_FromSupplement, FALSE);
		
END_CASE
END_METHOD

METHOD FB_init : BOOL
VAR_INPUT
	bInitRetains : BOOL; // if TRUE, the retain variables are initialized (warm start / cold start)
	bInCopyCode : BOOL;  // if TRUE, the instance afterwards gets moved into the copy code (online change)
END_VAR
eObjectType := E_BACnetObjType.ObjBinaryOutput;
END_METHOD

END_FUNCTION_BLOCK

// POUs/Local/Objects/[Base]/FB_BACnet_BaseMI
FUNCTION_BLOCK FB_BACnet_BaseMI EXTENDS FB_BACnet_EventObject
VAR_INPUT CONSTANT PERSISTENT
	{region 'Variable Parameters'}
		{attribute 'parameterCategory':='Value'}
		bEnOutOfService : BOOL;
		
		{attribute 'parameterCategory':='Hardware'}
		{attribute 'TcEncoding':='UTF-8'}
		sDeviceType : STRING;
	{endregion}
	{region 'Fixed Parameters'}
		{attribute 'parameterCategory':='Value'}
		{attribute 'TcEncoding':='UTF-8'}
		sStateText : ARRAY[1..BACnet_Param.nMultistate_StateCount] OF T_BACnet_StateText;
		
		{attribute 'parameterCategory':='EventConfig'}
		nAlarmValues : ARRAY[1..BACnet_Param.nMultistate_StateCount] OF UDINT;
		{attribute 'parameterCategory':='EventConfig'}
		nFaultValues : ARRAY[1..BACnet_Param.nMultistate_StateCount] OF UDINT;
	{endregion}
END_VAR
VAR_OUTPUT
	nPresentValue		: UDINT		:= 1;
END_VAR
VAR
	{region 'Output-Properties'}
		nStateCount		: UDINT;
	{endregion}
END_VAR

SUPER^();

METHOD PROTECTED OnObjectStateChanged
SUPER^.OnObjectStateChanged();

CASE (tState) OF
	TCOM_STATE.TCOM_STATE_PREOP:
		// SyncHandler:
		{warning disable C0196}
		nStateCount := F_BACnet_GetUsedStateText(sStateText);
		{warning restore C0196}
		
		RequestSyncHandlers(0, nStateCount);								// Handlers for "E_BACnetPropIdentifier.PropStateText"
		RequestSyncHandlers(0, F_BACnet_GetUsedUDINT(nAlarmValues));		// Handlers for "E_BACnetPropIdentifier.PropAlarmValues"
		RequestSyncHandlers(0, F_BACnet_GetUsedUDINT(nFaultValues));		// Handlers for "E_BACnetPropIdentifier.PropFaultValues"
		RequestSyncHandlers(0, 3);											// Handlers for other properties
		
		// Properties:
		WriteProtectProperty(E_BACnetPropIdentifier.PropNumberOfStates, TRUE);
		
		IF (BACnet_Param.bStateText_WriteProtect) THEN
			WriteProtectProperty(E_BACnetPropIdentifier.PropStateText, TRUE);
		END_IF
		
		// Ensure UTF-8 Encoding:
		F_BA_EnsureUTF8(ADR(sDeviceType), SIZEOF(sDeviceType));
		F_BA_EnsureUTF8Array(ADR(sStateText), SIZEOF(sStateText[1]), TO_DINT(BACnet_Param.nMultistate_StateCount));

	TCOM_STATE.TCOM_STATE_SAFEOP:
		SyncProperty(E_BACnetPropIdentifier.PropPresentValue, SIZEOF(nPresentValue), ADR(nPresentValue), 0, eSync_ToSupplement, TRUE);
		
	TCOM_STATE.TCOM_STATE_OP:
		// Init number of used states:
		SetNumberOfStates(nStateCount);
		
		SyncProperty(E_BACnetPropIdentifier.PropOutOfService, SIZEOF(bEnOutOfService), ADR(bEnOutOfService), 0, eFullSync_InitPLC, FALSE);
		SyncProperty(E_BACnetPropIdentifier.PropDeviceType, SIZEOF(sDeviceType), ADR(sDeviceType), 0, eFullSync_InitPLC, FALSE);
		SyncPropertyList(E_BACnetPropIdentifier.PropStateText, ADR(sStateText), SIZEOF(T_BACnet_StateText), nStateCount, eFullSync_InitPLC, FALSE);
		SyncPropertyList(E_BACnetPropIdentifier.PropAlarmValues, ADR(nAlarmValues), SIZEOF(UDINT), nStateCount, eFullSync_InitPLC, TRUE);
		SyncPropertyList(E_BACnetPropIdentifier.PropFaultValues, ADR(nFaultValues), SIZEOF(UDINT), nStateCount, eFullSync_InitPLC, TRUE);

END_CASE
END_METHOD

METHOD FB_init : BOOL
VAR_INPUT
	bInitRetains : BOOL; // if TRUE, the retain variables are initialized (warm start / cold start)
	bInCopyCode : BOOL;  // if TRUE, the instance afterwards gets moved into the copy code (online change)
END_VAR
eObjectType := E_BACnetObjType.ObjMultistateInput;
END_METHOD

PROPERTY StateCount : UDINT
GET
StateCount := nStateCount;
END_GET
END_PROPERTY

END_FUNCTION_BLOCK

// POUs/Local/Objects/[Base]/FB_BACnet_BaseMO
FUNCTION_BLOCK FB_BACnet_BaseMO EXTENDS FB_BACnet_EventObject
VAR_INPUT
	bEnPgm					: BOOL;
	nValPgm					: UDINT		:= 1;
END_VAR
VAR_INPUT CONSTANT PERSISTENT
	{region 'Variable Parameters'}
		{attribute 'parameterCategory':='Value'}
		nRelinquishDefault : UDINT := 1;
		{attribute 'parameterCategory':='Value'}
		bEnOutOfService : BOOL;
	
		{attribute 'parameterCategory':='Hardware'}
		{attribute 'TcEncoding':='UTF-8'}
		sDeviceType : STRING;
	{endregion}
	{region 'Fixed Parameters'}
		{attribute 'parameterCategory':='Value'}
		{attribute 'TcEncoding':='UTF-8'}
		sStateText : ARRAY[1..BACnet_Param.nMultistate_StateCount] OF T_BACnet_StateText;
	{endregion}
END_VAR
VAR_OUTPUT
	nPresentValue			: UDINT		:= 1;
END_VAR
VAR
	{region 'Output-Properties'}
		nStateCount			: UDINT;
	{endregion}
END_VAR
VAR
	{region 'Internal'}
		_nFeedbackValue		: UDINT;
	{endregion}
END_VAR

SUPER^();

METHOD PROTECTED OnObjectStateChanged
SUPER^.OnObjectStateChanged();

CASE (tState) OF
	TCOM_STATE.TCOM_STATE_PREOP:
		// SyncHandler:
		{warning disable C0196}
		nStateCount := F_BACnet_GetUsedStateText(sStateText);
		{warning restore C0196}
		
		RequestSyncHandlers(0, nStateCount);								// Handlers for "E_BACnetPropIdentifier.PropStateText"
		RequestSyncHandlers(1, 5);											// Handlers for other properties
		
		// Properties:
		WriteProtectProperty(E_BACnetPropIdentifier.PropNumberOfStates, TRUE);
		
		IF (BACnet_Param.bStateText_WriteProtect) THEN
			WriteProtectProperty(E_BACnetPropIdentifier.PropStateText, TRUE);
		END_IF
		
		// Ensure UTF-8 Encoding:
		F_BA_EnsureUTF8(ADR(sDeviceType), SIZEOF(sDeviceType));
		F_BA_EnsureUTF8Array(ADR(sStateText), SIZEOF(sStateText[1]), TO_DINT(BACnet_Param.nMultistate_StateCount));
		
	TCOM_STATE.TCOM_STATE_SAFEOP:
		SyncPropertyPvPrio(E_BACnetPropIdentifier.PropPresentValue, SIZEOF(nValPgm), ADR(nValPgm), ADR(bEnPgm), BACnet_Param.nPrio_Program, 0, eFullSync_InitPLC, TRUE);
		
		SyncProperty(E_BACnetPropIdentifier.PropPresentValue, SIZEOF(nPresentValue), ADR(nPresentValue), 0, eSync_FromSupplement, TRUE);
		
		SyncProperty(E_BACnetPropIdentifier.PropFeedbackValue, SIZEOF(_nFeedbackValue), ADR(_nFeedbackValue), 0, eSync_ToSupplement, TRUE);
		
	TCOM_STATE.TCOM_STATE_OP:
		// Init number of used states:
		SetNumberOfStates(nStateCount);
		
		SyncProperty(E_BACnetPropIdentifier.PropDeviceType, SIZEOF(sDeviceType), ADR(sDeviceType), 0, eFullSync_InitPLC, FALSE);
		SyncProperty(E_BACnetPropIdentifier.PropRelinquishDefault, SIZEOF(nRelinquishDefault), ADR(nRelinquishDefault), 0, eFullSync_InitPLC, FALSE);
		SyncProperty(E_BACnetPropIdentifier.PropOutOfService, SIZEOF(bEnOutOfService), ADR(bEnOutOfService), 0, eFullSync_InitPLC, FALSE);
		SyncPropertyList(E_BACnetPropIdentifier.PropStateText, ADR(sStateText), SIZEOF(T_BACnet_StateText), nStateCount, eFullSync_InitPLC, FALSE);
		
END_CASE
END_METHOD

METHOD FB_init : BOOL
VAR_INPUT
	bInitRetains : BOOL; // if TRUE, the retain variables are initialized (warm start / cold start)
	bInCopyCode : BOOL;  // if TRUE, the instance afterwards gets moved into the copy code (online change)
END_VAR
eObjectType := E_BACnetObjType.ObjMultistateOutput;
END_METHOD

PROPERTY StateCount : UDINT
GET
StateCount := nStateCount;
END_GET
END_PROPERTY

END_FUNCTION_BLOCK

// POUs/Local/Objects/[Base]/FB_BACnet_BaseSched
FUNCTION_BLOCK FB_BACnet_BaseSched EXTENDS FB_BACnet_Object
VAR_INPUT CONSTANT PERSISTENT
	{region 'Variable Parameters'}
		{attribute 'parameterCategory':='Value'}
		tWeek : T_BACnet_SchedWeek;															// Entries (separated per days) for weekly organization
		{attribute 'parameterCategory':='Value'}
		tCalendar : T_BACnet_SchedCalendar;													// Entries (separated per calendar) for global (calendar) exceptions organization (See "fbCalendar")
		{attribute 'parameterCategory':='Value'}
		tException : T_BACnet_SchedExceptionList;											// Entries (separated per exception count) for local (Presrent instance) exceptions organization
	{endregion}
END_VAR
VAR_INPUT CONSTANT
	{region 'Variable Parameters'}
		{attribute 'parameterCategory':='Value'}
		bWriteWeekly : BOOL;
		{attribute 'parameterCategory':='Value'}
		bWriteException : BOOL;
	{endregion}
END_VAR
VAR	
	{region 'COV'}
		bWeeklyChanged			: BOOL;
		bExceptionChanged		: BOOL;
	{endregion}
END_VAR
VAR
	{region 'Internal'}
		eDatatype				: E_BACnet_ValueChoice					:= E_BACnet_ValueChoice.eNullValue;
	{endregion}
END_VAR

IF (bWriteWeekly OR bWriteException) THEN
	WriteContent(bWriteWeekly, bWriteException);
	
	bWriteWeekly := FALSE;
	bWriteException := FALSE;
END_IF
IF (bWeeklyChanged OR bExceptionChanged) THEN
	ReadContent(bWeeklyChanged, bExceptionChanged);
	
	bWeeklyChanged := FALSE;
	bExceptionChanged := FALSE;
END_IF

SUPER^();

METHOD PROTECTED OnObjectStateChanged
SUPER^.OnObjectStateChanged();

CASE (tState) OF
	TCOM_STATE.TCOM_STATE_PREOP:
		// SyncHandler:
		RequestSyncHandlers(2, 0);
		
		// Properties:
		WriteProtectProperty(E_BACnetPropIdentifier.PropScheduleDefault, TRUE);
	
	TCOM_STATE.TCOM_STATE_SAFEOP:
		;
		
	TCOM_STATE.TCOM_STATE_OP:
		SyncPropertyCOV(bWeeklyChanged, E_BACnetPropIdentifier.PropWeeklySchedule);
		SyncPropertyCOV(bExceptionChanged, E_BACnetPropIdentifier.PropExceptionSchedule);
	
		WriteContent(TRUE, TRUE);
		WritePropertyUDInt(E_BACnetPropIdentifier.PropPriorityForWriting, BACnet_Param.nSched_PrioForWriting);
		
END_CASE
END_METHOD

METHOD FB_init : BOOL
VAR_INPUT
	bInitRetains : BOOL; // if TRUE, the retain variables are initialized (warm start / cold start)
	bInCopyCode : BOOL;  // if TRUE, the instance afterwards gets moved into the copy code (online change)
END_VAR
eObjectType := E_BACnetObjType.ObjSchedule;
END_METHOD

METHOD ReadContent : BOOL
VAR_INPUT
	bWeeklySched		: BOOL		:= TRUE;
	bExceptSched		: BOOL		:= TRUE;
END_VAR
IF bWeeklySched THEN
	IF (ReadPropertyWeeklySched(tWeek, eDataType) <> S_OK) THEN
		RETURN;
	END_IF
END_IF
IF bExceptSched THEN
	IF (ReadPropertyExceptionSched(tCalendar, tException, eDataType) <> S_OK) THEN
		RETURN;
	END_IF
END_IF

ReadContent := TRUE;
END_METHOD

METHOD WriteContent : BOOL
VAR_INPUT
	bWeeklySched		: BOOL		:= TRUE;
	bExceptSched		: BOOL		:= TRUE;
END_VAR
IF bWeeklySched THEN
	IF (WritePropertyWeeklySched(tWeek, eDataType) <> S_OK) THEN
		RETURN;
	END_IF
END_IF
IF bExceptSched THEN
	IF (WritePropertyExceptionSched(tCalendar, tException, eDataType) <> S_OK) THEN
		RETURN;
	END_IF
END_IF

WriteContent := TRUE;
END_METHOD

END_FUNCTION_BLOCK

// POUs/Local/Objects/[Base]/FB_BACnet_BaseTLog
FUNCTION_BLOCK FB_BACnet_BaseTLog EXTENDS FB_BACnet_EventObject
VAR_INPUT CONSTANT PERSISTENT
	{region 'Fixed Parameters'}
		{attribute 'parameterCategory':='Value'}
		nBufferSize : UDINT := BACnet_Param.nTLog_ArraySize;
	{endregion}
	{region 'Variable Parameters'}
		{attribute 'parameterCategory':='State'}
		bLogEnable : BOOL;
		
		{attribute 'parameterCategory':='Config'}
		stStartTime : ST_BA_DateTime;
		{attribute 'parameterCategory':='Config'}
		stStopTime : ST_BA_DateTime;
		{attribute 'parameterCategory':='Config'}
		bStopWhenFull : BOOL;
		{attribute 'parameterCategory':='Config'}
		{attribute 'parameterUnit':= '1/100s'}
		nLogInterval : UDINT := 9000;
		{attribute 'parameterCategory':='Config'}
		nNotificationThreshold : UDINT := 50;
		{attribute 'parameterCategory':='Config'}
		eLoggingType : E_BA_LoggingType := E_BA_LoggingType.ePolled;
	{endregion}
END_VAR
VAR_OUTPUT
	nRecordCount				: UDINT;
	nTotalRecordCount			: UDINT;
END_VAR

SUPER^();

METHOD PROTECTED OnObjectStateChanged
VAR
	_pBufferVal		: PVOID;
	_nBufferSize	: DINT;
END_VAR
SUPER^.OnObjectStateChanged();

CASE (tState) OF
	TCOM_STATE.TCOM_STATE_PREOP:
		// SyncHandler:
		RequestSyncHandlers(2, 7);
		
		// Properties:
		// May limit buffer size to respect array size:
		nBufferSize := MIN(BACnet_Param.nTLog_ArraySize, nBufferSize);
		
		WritePropertyUDInt(E_BACnetPropIdentifier.PropBufferSize, nBufferSize);
		
	TCOM_STATE.TCOM_STATE_SAFEOP:
		;

	TCOM_STATE.TCOM_STATE_OP:
		// Synchronize:
		SyncProperty(E_BACnetPropIdentifier.PropRecordCount, SIZEOF(nRecordCount), ADR(nRecordCount), 0, eSync_FromSupplement, FALSE);
		SyncProperty(E_BACnetPropIdentifier.PropTotalRecordCount, SIZEOF(nTotalRecordCount), ADR(nTotalRecordCount), 0, eSync_FromSupplement, FALSE);
		
		SyncProperty(E_BACnetPropIdentifier.PropEnable, SIZEOF(bLogEnable), ADR(bLogEnable), 0, eFullSync_InitPLC, FALSE);
		SyncProperty(E_BACnetPropIdentifier.PropStartTime, SIZEOF(stStartTime), ADR(stStartTime), 0, eFullSync_InitPLC, FALSE);
		SyncProperty(E_BACnetPropIdentifier.PropStopTime, SIZEOF(stStopTime), ADR(stStopTime), 0, eFullSync_InitPLC, FALSE);
		SyncProperty(E_BACnetPropIdentifier.PropStopWhenFull, SIZEOF(bStopWhenFull), ADR(bStopWhenFull), 0, eFullSync_InitPLC, FALSE);
		SyncProperty(E_BACnetPropIdentifier.PropLogInterval, SIZEOF(nLogInterval), ADR(nLogInterval), 0, eFullSync_InitPLC, FALSE);
		SyncProperty(E_BACnetPropIdentifier.PropNotificationThreshold, SIZEOF(nNotificationThreshold), ADR(nNotificationThreshold), 0, eFullSync_InitPLC, FALSE);
		SyncProperty(E_BACnetPropIdentifier.PropLoggingType, SIZEOF(eLoggingType), ADR(eLoggingType), 0, eFullSync_InitPLC, FALSE);
		
END_CASE
END_METHOD

END_FUNCTION_BLOCK

// POUs/Local/Objects/[Internal]/Property/Buffer/[Archiv]/FB_BACnet_WeeklyScheduleBuffer
FUNCTION_BLOCK INTERNAL FB_BACnet_WeeklyScheduleBuffer EXTENDS FB_BACnet_BaseListBuffer

SUPER^();

METHOD FB_init : BOOL
VAR_INPUT
	bInitRetains : BOOL; // if TRUE, the retain variables are initialized (warm start / cold start)
	bInCopyCode : BOOL;  // if TRUE, the instance afterwards gets moved into the copy code (online change)
END_VAR
ePropertyID := E_BACnetPropIdentifier.PropWeeklySchedule;
END_METHOD

METHOD ResetValue
VAR
	_nDay : INT;
END_VAR
SUPER^.ResetValue();

// Write empty weekday-array to buffer:
FOR _nDay := E_BA_Weekday.First TO E_BA_Weekday.Last DO
	MemSetULINT(16#0000000080000008, nUsedSize);
	MemSetULINT(16#0000000000000000, nUsedSize);
END_FOR

(*
FOR iDayTmp := iWeekdayFirst TO iWeekdayLast DO
	MemSetULINT(16#0000000080000020, nUsedSize);
	MemSetULINT(16#0000000000000000, nUsedSize);
	MemSetULINT(16#0000000000000000, nUsedSize);
	MemSetULINT(16#0000000000000000, nUsedSize);
	MemSetULINT(16#0000000000000000, nUsedSize);
END_FOR
*)
END_METHOD

END_FUNCTION_BLOCK

// POUs/Local/Objects/[Internal]/Property/Buffer/Base/FB_BACnet_BaseListBuffer
FUNCTION_BLOCK INTERNAL FB_BACnet_BaseListBuffer EXTENDS FB_BACnet_BasePropertyBuffer
VAR PERSISTENT
	bBuffer : ARRAY[1 .. nBACnet_BufferSize] OF BYTE;
END_VAR
VAR CONSTANT
	{attribute 'hide'}
	{attribute 'parameterUnit':= 'byte'}
	nBACnet_BufferSize	: UINT	:= 8192;
END_VAR

SUPER^();

METHOD PROTECTED ValidateInst : BOOL
nBufferSize := SIZEOF(bBuffer);
pBufferValue := ADR(bBuffer);

ValidateInst := SUPER^.ValidateInst();
END_METHOD

END_FUNCTION_BLOCK

// POUs/Local/Objects/[Internal]/Property/Buffer/Base/FB_BACnet_BasePropertyBuffer
FUNCTION_BLOCK INTERNAL FB_BACnet_BasePropertyBuffer
VAR_OUTPUT
	ePropertyID : E_BACnetPropIdentifier := E_BACnetPropIdentifier.PropInvalid;		// ID of referred property
	bChangeTrig : BOOL;												// Change trigger
	nChanges : UINT;												// Changes counter
	bIsReady : BOOL;												// Synchronization of referred property successfully initialized
END_VAR
VAR PERSISTENT
	nUsedSize : UDINT;
END_VAR
VAR
	// Init via instance-declaration:
	iRefObject : I_BACnet_Object;
	
	// Init via SubClass:
	tSyncState : TCOM_STATE := TCOM_STATE.TCOM_STATE_OP;						// Object-state to init synchronization of referred property
END_VAR
VAR_STAT
	// (BETA) ... Following symbols should be made non-static / thread safe!
	// Use "ValidateInst()" to ensure data to be valid: 
	fbRefObject : POINTER TO FB_BACnet_Object;
	nBufferSize : UDINT;
	pBufferValue : PVOID;
END_VAR
(*
VAR
	// [DEBUG]:
	eDebugCommand : (eNone:=1, eReadBuffer:=2, eWriteBuffer:=3, eResetBuffer:=4, ePrintBuffer:=5) UDINT := 1;
	sDebugHexBuffer : T_MaxString;
END_VAR
*)

IF (bChangeTrig) THEN
	bChangeTrig := FALSE;
	nChanges := (nChanges+1);
	
	IF (ValidateInst()) THEN
		// Refresh property value:
		ReadValue();
	END_IF
END_IF

(*
// [DEBUG]:
IF (eDebugCommand <> eNone) THEN
	IF (ValidateInst()) THEN
		CASE (eDebugCommand) OF
			eReadBuffer:
				ReadValue();
			eWriteBuffer:
				WriteValue();
			eResetBuffer:
				ResetValue();
			ePrintBuffer:
				sDebugHexBuffer := DATA_TO_HEXSTR(pData:=pBufferValue, cbData:=TO_UDINT(nUsedSize), FALSE);
		END_CASE
	END_IF
	eDebugCommand := eNone;
END_IF
*)

METHOD PRIVATE ReadValue : HRESULT
nUsedSize := nBufferSize;
ReadValue := fbRefObject^.ReadProperty(ePropertyID, pBufferValue, ADR(nUsedSize));
END_METHOD

METHOD PRIVATE WriteValue : HRESULT
WriteValue := fbRefObject^.WriteProperty(ePropertyID, pBufferValue, TO_DINT(nUsedSize));
END_METHOD

// Write a (any type) value to the memory buffer. 
// > Ensure to point to valid memory buffer via "ValidateInst()"!
METHOD PROTECTED MemSet : BOOL
VAR_INPUT
	xValue : ANY;
END_VAR
VAR_IN_OUT
	nOffset : UDINT;
END_VAR
VAR
	_nSizeTmp : UDINT;
END_VAR
_nSizeTmp := TO_UDINT(xValue.diSize);

IF (pBufferValue = 0) THEN
	F_BA_LogMessage(ADSLOG_MSGTYPE_ERROR, 'MS02', 'PropertyBuffer.MemSet: Uninitialized buffer!');
ELSIF ((_nSizeTmp+nOffset) > nBufferSize) THEN
	F_BA_LogMessage(ADSLOG_MSGTYPE_ERROR, 'MS04', 'PropertyBuffer.MemSet: Buffer size exceeded!');
ELSE
	MEMCPY((pBufferValue+nOffset), xValue.pValue, _nSizeTmp);
	nOffset := (nOffset+_nSizeTmp);
	
	MemSet := TRUE;
END_IF
END_METHOD

// Write a 1Byte-value to the memory buffer. 
METHOD PROTECTED MemSetBYTE : BOOL
VAR_INPUT
	nValue : BYTE;
END_VAR
VAR_IN_OUT
	nOffset : UDINT;
END_VAR
MemSetBYTE := MemSet(nValue, nOffset);
END_METHOD

// Write a 4Byte-value to the memory buffer. 
METHOD PROTECTED MemSetUDINT : BOOL
VAR_INPUT
	nValue : UDINT;
END_VAR
VAR_IN_OUT
	nOffset : UDINT;
END_VAR
MemSetUDINT := MemSet(nValue, nOffset);
END_METHOD

// Write a 2Byte-value to the memory buffer. 
METHOD PROTECTED MemSetUINT : BOOL
VAR_INPUT
	nValue : UINT;
END_VAR
VAR_IN_OUT
	nOffset : UDINT;
END_VAR
MemSetUINT := MemSet(nValue, nOffset);
END_METHOD

// Write a 8Byte-value to the memory buffer. 
METHOD PROTECTED MemSetULINT : BOOL
VAR_INPUT
	nValue : ULINT;
END_VAR
VAR_IN_OUT
	nOffset : UDINT;
END_VAR
MemSetULINT := MemSet(nValue, nOffset);
END_METHOD

METHOD PROTECTED ValidateInst : BOOL
IF (iRefObject = 0) THEN
	F_BA_LogMessage(ADSLOG_MSGTYPE_ERROR, 'GB3', 'PropertyBuffer: Unreferred object!');
	
ELSIF (NOT __QUERYPOINTER(iRefObject, fbRefObject)) OR (fbRefObject = 0) THEN
	F_BA_LogMessage(ADSLOG_MSGTYPE_ERROR, 'GB6', 'PropertyBuffer: Invalid referred object!');
	
ELSIF (nBufferSize = 0) OR (pBufferValue = 0) THEN
	F_BA_LogMessage1(ADSLOG_MSGTYPE_ERROR, 'GB8', 'PropertyBuffer: Unimplemented buffer of property "%d"!', F_INT(ePropertyID));

ELSE
	ValidateInst := TRUE;
END_IF
END_METHOD

METHOD OnObjectStateChanged
VAR_INPUT
	tState : TCOM_STATE;
END_VAR
VAR
	eSyncMode : E_BA_FullSyncMode := eFullSync_InitPLC;
END_VAR
IF (tState = tSyncState) THEN
	IF (ePropertyID = E_BACnetPropIdentifier.PropInvalid) THEN
		F_BA_LogMessage(ADSLOG_MSGTYPE_ERROR, 'OOSC8', 'PropertyBuffer: Uninitialized property type!');
		
	ELSIF (ValidateInst()) THEN
		// Initialize COV-Trigger:
		IF (fbRefObject^.SyncPropertyCOV(bChangeTrig, ePropertyID)) THEN
			// Initialize property:
			
			IF (nUsedSize = 0) THEN
				// Initial value has defenitly to be read from stack:
				bIsReady := SUCCEEDED(ReadValue());
			ELSE
				CASE (eSyncMode) OF
					eSync_ToSupplement,
					eFullSync_InitPLC:
						bIsReady := SUCCEEDED(WriteValue());
				ELSE
					bIsReady := SUCCEEDED(ReadValue());
				END_CASE
			END_IF
		END_IF
	END_IF
END_IF
END_METHOD

METHOD ResetValue
nUsedSize := 0;

ValidateInst();
END_METHOD

END_FUNCTION_BLOCK

// POUs/Local/Objects/[Internal]/Property/Buffer/Base/FB_BACnet_BaseArrayBuffer
FUNCTION_BLOCK INTERNAL FB_BACnet_BaseArrayBuffer EXTENDS FB_BACnet_BasePropertyBuffer
VAR CONSTANT
	{attribute 'hide'}
	nBACnet_EntryCount	: UINT	:= 256;
	
	// Hint:
	// > [BufferSize] := (nBACnet_EntryCount * [EntrySize])
END_VAR

SUPER^();

END_FUNCTION_BLOCK

// POUs/Local/Objects/[Internal]/Property/Buffer/FB_BACnet_DateListBuffer
FUNCTION_BLOCK INTERNAL FB_BACnet_DateListBuffer EXTENDS FB_BACnet_BaseListBuffer

SUPER^();

METHOD FB_init : BOOL
VAR_INPUT
	bInitRetains : BOOL; // if TRUE, the retain variables are initialized (warm start / cold start)
	bInCopyCode : BOOL;  // if TRUE, the instance afterwards gets moved into the copy code (online change)
END_VAR
ePropertyID := E_BACnetPropIdentifier.PropDateList;
END_METHOD

END_FUNCTION_BLOCK

// POUs/Local/Objects/[Internal]/Property/Buffer/FB_BACnet_EventLogBuffer
FUNCTION_BLOCK INTERNAL FB_BACnet_EventLogBuffer EXTENDS FB_BACnet_BasePropertyBuffer
VAR PERSISTENT
	bBuffer : ARRAY[1 .. nBACnet_BufferSize] OF BYTE;
END_VAR
VAR CONSTANT
	{attribute 'hide'}
	{attribute 'parameterUnit':= 'byte'}
	nBACnet_EntrySize	: UINT	:= 376;
	{attribute 'hide'}
	nBACnet_EntryCount	: UINT	:= BACnet_Globals.nDataField_MaxEventLogBufferEntries;
	
	{attribute 'hide'}
	nBACnet_BufferSize	: UINT	:= (nBACnet_EntrySize * nBACnet_EntryCount);
END_VAR

SUPER^();

METHOD PROTECTED ValidateInst : BOOL
nBufferSize := SIZEOF(bBuffer);
pBufferValue := ADR(bBuffer);

ValidateInst := SUPER^.ValidateInst();
END_METHOD

METHOD FB_init : BOOL
VAR_INPUT
	bInitRetains : BOOL; // if TRUE, the retain variables are initialized (warm start / cold start)
	bInCopyCode : BOOL;  // if TRUE, the instance afterwards gets moved into the copy code (online change)
END_VAR
ePropertyID := E_BACnetPropIdentifier.PropLogBuffer;
END_METHOD

END_FUNCTION_BLOCK

// POUs/Local/Objects/[Internal]/Property/Buffer/FB_BACnet_ExceptionScheduleBuffer
FUNCTION_BLOCK INTERNAL FB_BACnet_ExceptionScheduleBuffer EXTENDS FB_BACnet_BaseListBuffer

SUPER^();

METHOD FB_init : BOOL
VAR_INPUT
	bInitRetains : BOOL; // if TRUE, the retain variables are initialized (warm start / cold start)
	bInCopyCode : BOOL;  // if TRUE, the instance afterwards gets moved into the copy code (online change)
END_VAR
ePropertyID := E_BACnetPropIdentifier.PropExceptionSchedule;
END_METHOD

END_FUNCTION_BLOCK

// POUs/Local/Objects/[Internal]/Property/Buffer/FB_BACnet_TLMBuffer
FUNCTION_BLOCK INTERNAL FB_BACnet_TLMBuffer EXTENDS FB_BACnet_BasePropertyBuffer
VAR PERSISTENT
	bBuffer : ARRAY[1 .. nBACnet_BufferSize] OF BYTE;
END_VAR
VAR CONSTANT
	{attribute 'hide'}
	{attribute 'parameterUnit':= 'byte'}
	nBACnet_HeaderSize		: UINT	:= 20;
	{attribute 'hide'}
	{attribute 'parameterUnit':= 'byte'}
	nBACnet_EntrySize		: UINT	:= 5;
	{attribute 'hide'}
	nBACnet_EntryCount		: UINT	:= BACnet_Globals.nDataField_MaxLogBufferEntries;
	{attribute 'hide'}
	nBACnet_EntryItemCount	: UINT	:= 100;
	
	{attribute 'hide'}
	nBACnet_BufferSize		: UINT	:= nBACnet_HeaderSize + ((nBACnet_EntrySize * nBACnet_EntryCount) * nBACnet_EntryItemCount);
END_VAR

SUPER^();

METHOD PROTECTED ValidateInst : BOOL
nBufferSize := SIZEOF(bBuffer);
pBufferValue := ADR(bBuffer);

ValidateInst := SUPER^.ValidateInst();
END_METHOD

METHOD FB_init : BOOL
VAR_INPUT
	bInitRetains : BOOL; // if TRUE, the retain variables are initialized (warm start / cold start)
	bInCopyCode : BOOL;  // if TRUE, the instance afterwards gets moved into the copy code (online change)
END_VAR
ePropertyID := E_BACnetPropIdentifier.PropLogBuffer;
END_METHOD

METHOD ResetValue
VAR
	stTimestamp : POINTER TO ST_BA_DateTime;
END_VAR
SUPER^.ResetValue();

// Write one log-entry "log-disabled" to buffer:
MemSetULINT(16#0000000100000020, nUsedSize);
MemSetUDINT(16#00000003, nUsedSize);

(*
stTimestamp := (pBufferValue+nUsedSize);
stTimestamp^ := F_GetCurrentTime();
nUsedSize := (nUsedSize+SIZEOF(ST_DateTime));
*)
MemSetULINT(16#51152607021D0177, nUsedSize);

MemSetUDINT(16#00000000, nUsedSize);
MemSetULINT(16#0000000000000008, nUsedSize);
MemSetULINT(16#0000800500000000, nUsedSize);
END_METHOD

END_FUNCTION_BLOCK

// POUs/Local/Objects/[Internal]/Property/Buffer/FB_BACnet_TrendLogBuffer
FUNCTION_BLOCK INTERNAL FB_BACnet_TrendLogBuffer EXTENDS FB_BACnet_BasePropertyBuffer
VAR PERSISTENT
	bBuffer : ARRAY[1 .. nBACnet_BufferSize] OF BYTE;
END_VAR
VAR CONSTANT
	{attribute 'hide'}
	{attribute 'parameterUnit':= 'byte'}
	nBACnet_EntrySize	: UINT	:= 56;
	{attribute 'hide'}
	nBACnet_EntryCount	: UINT	:= BACnet_Globals.nDataField_MaxLogBufferEntries;
	
	{attribute 'hide'}
	nBACnet_BufferSize	: UINT	:= (nBACnet_EntrySize * nBACnet_EntryCount);
END_VAR

SUPER^();

METHOD PROTECTED ValidateInst : BOOL
nBufferSize := SIZEOF(bBuffer);
pBufferValue := ADR(bBuffer);

ValidateInst := SUPER^.ValidateInst();
END_METHOD

METHOD FB_init : BOOL
VAR_INPUT
	bInitRetains : BOOL; // if TRUE, the retain variables are initialized (warm start / cold start)
	bInCopyCode : BOOL;  // if TRUE, the instance afterwards gets moved into the copy code (online change)
END_VAR
ePropertyID := E_BACnetPropIdentifier.PropLogBuffer;
END_METHOD

METHOD ResetValue
VAR
	stTimestamp : POINTER TO ST_BA_DateTime;
END_VAR
SUPER^.ResetValue();

// Write one log-entry "log-disabled" to buffer:
MemSetULINT(16#0000000100000020, nUsedSize);
MemSetUDINT(16#00000003, nUsedSize);

(*
stTimestamp := (pBufferValue+nUsedSize);
stTimestamp^ := F_GetCurrentTime();
nUsedSize := (nUsedSize+SIZEOF(ST_DateTime));
*)
MemSetULINT(16#51152607021D0177, nUsedSize);

MemSetUDINT(16#00000000, nUsedSize);
MemSetULINT(16#0000000000000008, nUsedSize);
MemSetULINT(16#0000800500000000, nUsedSize);
END_METHOD

END_FUNCTION_BLOCK

// POUs/Local/Objects/5P/FB_BACnet_AO_IO5P
// Analog Output Object
// - Terminal communication
// - 5 Priorities
FUNCTION_BLOCK FB_BACnet_AO_IO5P EXTENDS FB_BACnet_AO_IO
VAR_INPUT
	bEnSfty					: BOOL;
	fValSfty				: REAL;
	bEnCrit					: BOOL;
	fValCrit				: REAL;
	bEnManLoc				: BOOL;
	fValManLoc				: REAL;
END_VAR
VAR_INPUT CONSTANT PERSISTENT
	{region 'Operational Parameters'}
		{attribute 'parameterCategory':='Manual'}
		bEnManualRm : BOOL;
		{attribute 'parameterCategory':='Manual'}
		fValManualRm : REAL;
	{endregion}
END_VAR
VAR_OUTPUT
	nActivePrio				: UDINT;			// Indicates the currently active priority of the priority array
END_VAR

SUPER^();

METHOD PROTECTED OnObjectStateChanged
SUPER^.OnObjectStateChanged();

CASE (tState) OF
	TCOM_STATE.TCOM_STATE_PREOP:
		// SyncHandler:
		RequestSyncHandlers(1, 4);
		
	TCOM_STATE.TCOM_STATE_SAFEOP:
		SyncProperty(E_BACnetPropIdentifier.PropCurrentlyActivePriority, SIZEOF(nActivePrio), ADR(nActivePrio), 0, eSync_FromSupplement, TRUE);

		SyncPropertyPvPrio(E_BACnetPropIdentifier.PropPresentValue, SIZEOF(fValSfty), ADR(fValSfty), ADR(bEnSfty), BACnet_Param.nPrio_LifeSafety, 0, eFullSync_InitPLC, TRUE);
		SyncPropertyPvPrio(E_BACnetPropIdentifier.PropPresentValue, SIZEOF(fValCrit), ADR(fValCrit), ADR(bEnCrit), BACnet_Param.nPrio_Critical, 0, eFullSync_InitPLC, TRUE);
		SyncPropertyPvPrio(E_BACnetPropIdentifier.PropPresentValue, SIZEOF(fValManLoc), ADR(fValManLoc), ADR(bEnManLoc), BACnet_Param.nPrio_ManLocal, 0, eFullSync_InitPLC, TRUE);
		SyncPropertyPvPrio(E_BACnetPropIdentifier.PropPresentValue, SIZEOF(fValManualRm), ADR(fValManualRm), ADR(bEnManualRm), BACnet_Param.nPrio_ManRemote, 0, eFullSync_InitPLC, TRUE);
		
	TCOM_STATE.TCOM_STATE_OP:
		;
	
END_CASE
END_METHOD

PROPERTY ActivePrio : UDINT
GET
ActivePrio := nActivePrio;
END_GET
END_PROPERTY

PROPERTY EnManualRm : BOOL
GET
EnManualRm := bEnManualRm;
END_GET
SET
bEnManualRm := EnManualRm;
END_SET
END_PROPERTY

PROPERTY ValManualRm : REAL
GET
ValManualRm := fValManualRm;
END_GET
SET
fValManualRm := ValManualRm;
END_SET
END_PROPERTY

END_FUNCTION_BLOCK

// POUs/Local/Objects/FB_BACnet_AO_IO
// Analog Output Object
// - Terminal communication
// - 1 Priority
FUNCTION_BLOCK FB_BACnet_AO_IO EXTENDS FB_BACnet_BaseAO
VAR_INPUT CONSTANT PERSISTENT
	{region 'Variable Parameters'}
		{attribute 'parameterCategory':='Config'}
		eOverriddenPolarity : E_BA_Polarity := E_BA_Polarity.eNormal;
	{endregion}
END_VAR
VAR
	{region 'Raw I/O'}
		bRawOverridden		AT %I*	: BOOL;				// Raw overridden (Optional)
		nRawState			AT %I*	: USINT;			// Raw state (Optional, only used to determine overridden state)
		nRawValue			AT %Q*	: INT;				// Raw value
	{endregion}
	{region 'Hardware'}
		_bIsOverriddenMapped		: BOOL;				// Indication to mapped hardware for overridden IO value
		_bIsStateMapped				: BOOL;				// Indication to mapped hardware for state
	{endregion}
END_VAR

IF (bReady) THEN
	// Overridden IO Value:
	IF (_bIsOverriddenMapped) THEN
		_bOverriddenValue := (bRawOverridden = (eOverriddenPolarity=E_BA_Polarity.eNormal));
	ELSIF (_bIsStateMapped) THEN
		_bOverriddenValue := ((nRawState=0) = (eOverriddenPolarity=E_BA_Polarity.eNormal));
	ELSE
		_bOverriddenValue := FALSE;
	END_IF
END_IF

SUPER^();

METHOD PROTECTED OnObjectStateChanged
SUPER^.OnObjectStateChanged();

CASE (tState) OF
	TCOM_STATE.TCOM_STATE_PREOP:
		// SyncHandler:
		RequestSyncHandlers(1, 0);

	TCOM_STATE.TCOM_STATE_SAFEOP:
		SyncProperty(E_BACnetPropIdentifier.PropRawIoAnalogValueINT, SIZEOF(nRawValue), ADR(nRawValue), 0, eSync_FromSupplement, TRUE);
		
